BEGIN
   BB_G1.E.Ein := TRUE;
   BB_G1.E.Anst := FALSE;
   BB_G1.E.FU := FALSE;
   BB_G1.E.EA := FALSE;
   BB_G1.E.EZ := FALSE;
   BB_G1.E.MS_St := FALSE;
   BB_G1.E.Th_St := FALSE;
   BB_G1.E.DMA_St := FALSE;
   BB_G1.E.DMZ_St := FALSE;
   BB_G1.E.FU_St := FALSE;
   BB_G1.E.TL_St := FALSE;
   BB_G1.E.UDr_St := FALSE;
   BB_G1.E.UeDr_St := FALSE;
   BB_G1.E.UT_St := FALSE;
   BB_G1.E.Le_St := FALSE;
   BB_G1.E.UeLM_St := FALSE;
   BB_G1.E.UeLE_St := FALSE;
   BB_G1.E.Kom_DP_St := FALSE;
   BB_G1.E.Kom_int_St := FALSE;
   BB_G1.E.int_St := FALSE;
   BB_G1.E.Wart_Wa := FALSE;
   BB_G1.E.Bed_vOrt := FALSE;
   BB_G1.E.Bed_Fern := TRUE;
   BB_G1.E.Bed_UV := FALSE;
   BB_G1.E.Aus := FALSE;
   BB_G1.E.NA := FALSE;
   BB_G1.E.AF_St := FALSE;
   BB_G1.E.Strm := FALSE;
   BB_G1.E.FI_St := FALSE;
   BB_G1.E.SA_St := FALSE;
   BB_G1.E.DD_St := FALSE;
   BB_G1.E.St := FALSE;
   BB_G1.A.Ein := TRUE;
   BB_G1.A.B2 := FALSE;
   BB_G1.A.FU := FALSE;
   BB_G1.A.Req_extern_B1 := TRUE;
   BB_G1.A.Req_extern_B2 := FALSE;
   BB_G1.A.Dir := FALSE;
   BB_G1.A.RST := FALSE;
   BB_G1.A.Auf := FALSE;
   BB_G1.A.Zu := FALSE;
   BB_G1.A.Res9 := FALSE;
   BB_G1.A.Res10 := FALSE;
   BB_G1.A.Res11 := FALSE;
   BB_G1.A.Res12 := FALSE;
   BB_G1.A.Res13 := FALSE;
   BB_G1.A.Res14 := FALSE;
   BB_G1.A.Quit_extern := FALSE;
   BB_G2.E.Ein := TRUE;
   BB_G2.E.Anst := FALSE;
   BB_G2.E.FU := FALSE;
   BB_G2.E.EA := FALSE;
   BB_G2.E.EZ := FALSE;
   BB_G2.E.MS_St := FALSE;
   BB_G2.E.Th_St := FALSE;
   BB_G2.E.DMA_St := FALSE;
   BB_G2.E.DMZ_St := FALSE;
   BB_G2.E.FU_St := FALSE;
   BB_G2.E.TL_St := FALSE;
   BB_G2.E.UDr_St := FALSE;
   BB_G2.E.UeDr_St := FALSE;
   BB_G2.E.UT_St := FALSE;
   BB_G2.E.Le_St := FALSE;
   BB_G2.E.UeLM_St := FALSE;
   BB_G2.E.UeLE_St := FALSE;
   BB_G2.E.Kom_DP_St := FALSE;
   BB_G2.E.Kom_int_St := FALSE;
   BB_G2.E.int_St := FALSE;
   BB_G2.E.Wart_Wa := FALSE;
   BB_G2.E.Bed_vOrt := FALSE;
   BB_G2.E.Bed_Fern := TRUE;
   BB_G2.E.Bed_UV := FALSE;
   BB_G2.E.Aus := FALSE;
   BB_G2.E.NA := FALSE;
   BB_G2.E.AF_St := FALSE;
   BB_G2.E.Strm := FALSE;
   BB_G2.E.FI_St := FALSE;
   BB_G2.E.SA_St := FALSE;
   BB_G2.E.DD_St := FALSE;
   BB_G2.E.St := FALSE;
   BB_G2.A.Ein := TRUE;
   BB_G2.A.B2 := FALSE;
   BB_G2.A.FU := FALSE;
   BB_G2.A.Req_extern_B1 := TRUE;
   BB_G2.A.Req_extern_B2 := FALSE;
   BB_G2.A.Dir := FALSE;
   BB_G2.A.RST := FALSE;
   BB_G2.A.Auf := FALSE;
   BB_G2.A.Zu := FALSE;
   BB_G2.A.Res9 := FALSE;
   BB_G2.A.Res10 := FALSE;
   BB_G2.A.Res11 := FALSE;
   BB_G2.A.Res12 := FALSE;
   BB_G2.A.Res13 := FALSE;
   BB_G2.A.Res14 := FALSE;
   BB_G2.A.Quit_extern := FALSE;
   BB_G3.E.Ein := FALSE;
   BB_G3.E.Anst := FALSE;
   BB_G3.E.FU := FALSE;
   BB_G3.E.EA := FALSE;
   BB_G3.E.EZ := FALSE;
   BB_G3.E.MS_St := FALSE;
   BB_G3.E.Th_St := FALSE;
   BB_G3.E.DMA_St := FALSE;
   BB_G3.E.DMZ_St := FALSE;
   BB_G3.E.FU_St := FALSE;
   BB_G3.E.TL_St := FALSE;
   BB_G3.E.UDr_St := FALSE;
   BB_G3.E.UeDr_St := FALSE;
   BB_G3.E.UT_St := FALSE;
   BB_G3.E.Le_St := FALSE;
   BB_G3.E.UeLM_St := FALSE;
   BB_G3.E.UeLE_St := FALSE;
   BB_G3.E.Kom_DP_St := FALSE;
   BB_G3.E.Kom_int_St := FALSE;
   BB_G3.E.int_St := FALSE;
   BB_G3.E.Wart_Wa := FALSE;
   BB_G3.E.Bed_vOrt := FALSE;
   BB_G3.E.Bed_Fern := TRUE;
   BB_G3.E.Bed_UV := FALSE;
   BB_G3.E.Aus := FALSE;
   BB_G3.E.NA := FALSE;
   BB_G3.E.AF_St := FALSE;
   BB_G3.E.Strm := FALSE;
   BB_G3.E.FI_St := FALSE;
   BB_G3.E.SA_St := FALSE;
   BB_G3.E.DD_St := FALSE;
   BB_G3.E.St := FALSE;
   BB_G3.A.Ein := FALSE;
   BB_G3.A.B2 := FALSE;
   BB_G3.A.FU := FALSE;
   BB_G3.A.Req_extern_B1 := FALSE;
   BB_G3.A.Req_extern_B2 := FALSE;
   BB_G3.A.Dir := FALSE;
   BB_G3.A.RST := FALSE;
   BB_G3.A.Auf := FALSE;
   BB_G3.A.Zu := FALSE;
   BB_G3.A.Res9 := FALSE;
   BB_G3.A.Res10 := FALSE;
   BB_G3.A.Res11 := FALSE;
   BB_G3.A.Res12 := FALSE;
   BB_G3.A.Res13 := FALSE;
   BB_G3.A.Res14 := FALSE;
   BB_G3.A.Quit_extern := FALSE;
   BB_SHL_G1.E.Ein := TRUE;
   BB_SHL_G1.E.Anst := FALSE;
   BB_SHL_G1.E.FU := FALSE;
   BB_SHL_G1.E.EA := FALSE;
   BB_SHL_G1.E.EZ := FALSE;
   BB_SHL_G1.E.MS_St := FALSE;
   BB_SHL_G1.E.Th_St := FALSE;
   BB_SHL_G1.E.DMA_St := FALSE;
   BB_SHL_G1.E.DMZ_St := FALSE;
   BB_SHL_G1.E.FU_St := FALSE;
   BB_SHL_G1.E.TL_St := FALSE;
   BB_SHL_G1.E.UDr_St := FALSE;
   BB_SHL_G1.E.UeDr_St := FALSE;
   BB_SHL_G1.E.UT_St := FALSE;
   BB_SHL_G1.E.Le_St := FALSE;
   BB_SHL_G1.E.UeLM_St := FALSE;
   BB_SHL_G1.E.UeLE_St := FALSE;
   BB_SHL_G1.E.Kom_DP_St := FALSE;
   BB_SHL_G1.E.Kom_int_St := FALSE;
   BB_SHL_G1.E.int_St := FALSE;
   BB_SHL_G1.E.Wart_Wa := FALSE;
   BB_SHL_G1.E.Bed_vOrt := FALSE;
   BB_SHL_G1.E.Bed_Fern := TRUE;
   BB_SHL_G1.E.Bed_UV := FALSE;
   BB_SHL_G1.E.Aus := FALSE;
   BB_SHL_G1.E.NA := FALSE;
   BB_SHL_G1.E.AF_St := FALSE;
   BB_SHL_G1.E.Strm := FALSE;
   BB_SHL_G1.E.FI_St := FALSE;
   BB_SHL_G1.E.SA_St := FALSE;
   BB_SHL_G1.E.DD_St := FALSE;
   BB_SHL_G1.E.St := FALSE;
   BB_SHL_G1.A.Ein := FALSE;
   BB_SHL_G1.A.B2 := FALSE;
   BB_SHL_G1.A.FU := FALSE;
   BB_SHL_G1.A.Req_extern_B1 := FALSE;
   BB_SHL_G1.A.Req_extern_B2 := FALSE;
   BB_SHL_G1.A.Dir := FALSE;
   BB_SHL_G1.A.RST := FALSE;
   BB_SHL_G1.A.Auf := FALSE;
   BB_SHL_G1.A.Zu := FALSE;
   BB_SHL_G1.A.Res9 := FALSE;
   BB_SHL_G1.A.Res10 := FALSE;
   BB_SHL_G1.A.Res11 := FALSE;
   BB_SHL_G1.A.Res12 := FALSE;
   BB_SHL_G1.A.Res13 := FALSE;
   BB_SHL_G1.A.Res14 := FALSE;
   BB_SHL_G1.A.Quit_extern := FALSE;
   BB_SHL_G2.E.Ein := TRUE;
   BB_SHL_G2.E.Anst := FALSE;
   BB_SHL_G2.E.FU := FALSE;
   BB_SHL_G2.E.EA := FALSE;
   BB_SHL_G2.E.EZ := FALSE;
   BB_SHL_G2.E.MS_St := FALSE;
   BB_SHL_G2.E.Th_St := FALSE;
   BB_SHL_G2.E.DMA_St := FALSE;
   BB_SHL_G2.E.DMZ_St := FALSE;
   BB_SHL_G2.E.FU_St := FALSE;
   BB_SHL_G2.E.TL_St := FALSE;
   BB_SHL_G2.E.UDr_St := FALSE;
   BB_SHL_G2.E.UeDr_St := FALSE;
   BB_SHL_G2.E.UT_St := FALSE;
   BB_SHL_G2.E.Le_St := FALSE;
   BB_SHL_G2.E.UeLM_St := FALSE;
   BB_SHL_G2.E.UeLE_St := FALSE;
   BB_SHL_G2.E.Kom_DP_St := FALSE;
   BB_SHL_G2.E.Kom_int_St := FALSE;
   BB_SHL_G2.E.int_St := FALSE;
   BB_SHL_G2.E.Wart_Wa := FALSE;
   BB_SHL_G2.E.Bed_vOrt := FALSE;
   BB_SHL_G2.E.Bed_Fern := TRUE;
   BB_SHL_G2.E.Bed_UV := FALSE;
   BB_SHL_G2.E.Aus := FALSE;
   BB_SHL_G2.E.NA := FALSE;
   BB_SHL_G2.E.AF_St := FALSE;
   BB_SHL_G2.E.Strm := FALSE;
   BB_SHL_G2.E.FI_St := FALSE;
   BB_SHL_G2.E.SA_St := FALSE;
   BB_SHL_G2.E.DD_St := FALSE;
   BB_SHL_G2.E.St := FALSE;
   BB_SHL_G2.A.Ein := FALSE;
   BB_SHL_G2.A.B2 := FALSE;
   BB_SHL_G2.A.FU := FALSE;
   BB_SHL_G2.A.Req_extern_B1 := FALSE;
   BB_SHL_G2.A.Req_extern_B2 := FALSE;
   BB_SHL_G2.A.Dir := FALSE;
   BB_SHL_G2.A.RST := FALSE;
   BB_SHL_G2.A.Auf := FALSE;
   BB_SHL_G2.A.Zu := FALSE;
   BB_SHL_G2.A.Res9 := FALSE;
   BB_SHL_G2.A.Res10 := FALSE;
   BB_SHL_G2.A.Res11 := FALSE;
   BB_SHL_G2.A.Res12 := FALSE;
   BB_SHL_G2.A.Res13 := FALSE;
   BB_SHL_G2.A.Res14 := FALSE;
   BB_SHL_G2.A.Quit_extern := FALSE;
   BB_SHL_G3.E.Ein := FALSE;
   BB_SHL_G3.E.Anst := FALSE;
   BB_SHL_G3.E.FU := FALSE;
   BB_SHL_G3.E.EA := FALSE;
   BB_SHL_G3.E.EZ := FALSE;
   BB_SHL_G3.E.MS_St := FALSE;
   BB_SHL_G3.E.Th_St := FALSE;
   BB_SHL_G3.E.DMA_St := FALSE;
   BB_SHL_G3.E.DMZ_St := FALSE;
   BB_SHL_G3.E.FU_St := FALSE;
   BB_SHL_G3.E.TL_St := FALSE;
   BB_SHL_G3.E.UDr_St := FALSE;
   BB_SHL_G3.E.UeDr_St := FALSE;
   BB_SHL_G3.E.UT_St := FALSE;
   BB_SHL_G3.E.Le_St := FALSE;
   BB_SHL_G3.E.UeLM_St := FALSE;
   BB_SHL_G3.E.UeLE_St := FALSE;
   BB_SHL_G3.E.Kom_DP_St := FALSE;
   BB_SHL_G3.E.Kom_int_St := FALSE;
   BB_SHL_G3.E.int_St := FALSE;
   BB_SHL_G3.E.Wart_Wa := FALSE;
   BB_SHL_G3.E.Bed_vOrt := FALSE;
   BB_SHL_G3.E.Bed_Fern := TRUE;
   BB_SHL_G3.E.Bed_UV := FALSE;
   BB_SHL_G3.E.Aus := FALSE;
   BB_SHL_G3.E.NA := FALSE;
   BB_SHL_G3.E.AF_St := FALSE;
   BB_SHL_G3.E.Strm := FALSE;
   BB_SHL_G3.E.FI_St := FALSE;
   BB_SHL_G3.E.SA_St := FALSE;
   BB_SHL_G3.E.DD_St := FALSE;
   BB_SHL_G3.E.St := FALSE;
   BB_SHL_G3.A.Ein := FALSE;
   BB_SHL_G3.A.B2 := FALSE;
   BB_SHL_G3.A.FU := FALSE;
   BB_SHL_G3.A.Req_extern_B1 := FALSE;
   BB_SHL_G3.A.Req_extern_B2 := FALSE;
   BB_SHL_G3.A.Dir := FALSE;
   BB_SHL_G3.A.RST := FALSE;
   BB_SHL_G3.A.Auf := FALSE;
   BB_SHL_G3.A.Zu := FALSE;
   BB_SHL_G3.A.Res9 := FALSE;
   BB_SHL_G3.A.Res10 := FALSE;
   BB_SHL_G3.A.Res11 := FALSE;
   BB_SHL_G3.A.Res12 := FALSE;
   BB_SHL_G3.A.Res13 := FALSE;
   BB_SHL_G3.A.Res14 := FALSE;
   BB_SHL_G3.A.Quit_extern := FALSE;
   BB_AV.E.Ein := FALSE;
   BB_AV.E.Anst := FALSE;
   BB_AV.E.FU := FALSE;
   BB_AV.E.EA := FALSE;
   BB_AV.E.EZ := FALSE;
   BB_AV.E.MS_St := FALSE;
   BB_AV.E.Th_St := FALSE;
   BB_AV.E.DMA_St := FALSE;
   BB_AV.E.DMZ_St := FALSE;
   BB_AV.E.FU_St := FALSE;
   BB_AV.E.TL_St := FALSE;
   BB_AV.E.UDr_St := FALSE;
   BB_AV.E.UeDr_St := FALSE;
   BB_AV.E.UT_St := FALSE;
   BB_AV.E.Le_St := FALSE;
   BB_AV.E.UeLM_St := FALSE;
   BB_AV.E.UeLE_St := FALSE;
   BB_AV.E.Kom_DP_St := FALSE;
   BB_AV.E.Kom_int_St := FALSE;
   BB_AV.E.int_St := FALSE;
   BB_AV.E.Wart_Wa := FALSE;
   BB_AV.E.Bed_vOrt := FALSE;
   BB_AV.E.Bed_Fern := TRUE;
   BB_AV.E.Bed_UV := FALSE;
   BB_AV.E.Aus := FALSE;
   BB_AV.E.NA := FALSE;
   BB_AV.E.AF_St := FALSE;
   BB_AV.E.Strm := FALSE;
   BB_AV.E.FI_St := FALSE;
   BB_AV.E.SA_St := FALSE;
   BB_AV.E.DD_St := FALSE;
   BB_AV.E.St := FALSE;
   BB_AV.A.Ein := FALSE;
   BB_AV.A.B2 := FALSE;
   BB_AV.A.FU := FALSE;
   BB_AV.A.Req_extern_B1 := FALSE;
   BB_AV.A.Req_extern_B2 := FALSE;
   BB_AV.A.Dir := FALSE;
   BB_AV.A.RST := FALSE;
   BB_AV.A.Auf := FALSE;
   BB_AV.A.Zu := FALSE;
   BB_AV.A.Res9 := FALSE;
   BB_AV.A.Res10 := FALSE;
   BB_AV.A.Res11 := FALSE;
   BB_AV.A.Res12 := FALSE;
   BB_AV.A.Res13 := FALSE;
   BB_AV.A.Res14 := FALSE;
   BB_AV.A.Quit_extern := FALSE;
   BB_LS1.E.Ein := FALSE;
   BB_LS1.E.Anst := FALSE;
   BB_LS1.E.FU := FALSE;
   BB_LS1.E.EA := FALSE;
   BB_LS1.E.EZ := TRUE;
   BB_LS1.E.MS_St := FALSE;
   BB_LS1.E.Th_St := FALSE;
   BB_LS1.E.DMA_St := FALSE;
   BB_LS1.E.DMZ_St := FALSE;
   BB_LS1.E.FU_St := FALSE;
   BB_LS1.E.TL_St := FALSE;
   BB_LS1.E.UDr_St := FALSE;
   BB_LS1.E.UeDr_St := FALSE;
   BB_LS1.E.UT_St := FALSE;
   BB_LS1.E.Le_St := FALSE;
   BB_LS1.E.UeLM_St := FALSE;
   BB_LS1.E.UeLE_St := FALSE;
   BB_LS1.E.Kom_DP_St := FALSE;
   BB_LS1.E.Kom_int_St := FALSE;
   BB_LS1.E.int_St := FALSE;
   BB_LS1.E.Wart_Wa := FALSE;
   BB_LS1.E.Bed_vOrt := FALSE;
   BB_LS1.E.Bed_Fern := TRUE;
   BB_LS1.E.Bed_UV := FALSE;
   BB_LS1.E.Aus := FALSE;
   BB_LS1.E.NA := FALSE;
   BB_LS1.E.AF_St := FALSE;
   BB_LS1.E.Strm := FALSE;
   BB_LS1.E.FI_St := FALSE;
   BB_LS1.E.SA_St := FALSE;
   BB_LS1.E.DD_St := FALSE;
   BB_LS1.E.St := FALSE;
   BB_LS1.A.Ein := FALSE;
   BB_LS1.A.B2 := FALSE;
   BB_LS1.A.FU := FALSE;
   BB_LS1.A.Req_extern_B1 := FALSE;
   BB_LS1.A.Req_extern_B2 := FALSE;
   BB_LS1.A.Dir := FALSE;
   BB_LS1.A.RST := FALSE;
   BB_LS1.A.Auf := FALSE;
   BB_LS1.A.Zu := FALSE;
   BB_LS1.A.Res9 := FALSE;
   BB_LS1.A.Res10 := FALSE;
   BB_LS1.A.Res11 := FALSE;
   BB_LS1.A.Res12 := FALSE;
   BB_LS1.A.Res13 := FALSE;
   BB_LS1.A.Res14 := FALSE;
   BB_LS1.A.Quit_extern := FALSE;
   BB_LS2.E.Ein := FALSE;
   BB_LS2.E.Anst := FALSE;
   BB_LS2.E.FU := FALSE;
   BB_LS2.E.EA := FALSE;
   BB_LS2.E.EZ := TRUE;
   BB_LS2.E.MS_St := FALSE;
   BB_LS2.E.Th_St := FALSE;
   BB_LS2.E.DMA_St := FALSE;
   BB_LS2.E.DMZ_St := FALSE;
   BB_LS2.E.FU_St := FALSE;
   BB_LS2.E.TL_St := FALSE;
   BB_LS2.E.UDr_St := FALSE;
   BB_LS2.E.UeDr_St := FALSE;
   BB_LS2.E.UT_St := FALSE;
   BB_LS2.E.Le_St := FALSE;
   BB_LS2.E.UeLM_St := FALSE;
   BB_LS2.E.UeLE_St := FALSE;
   BB_LS2.E.Kom_DP_St := FALSE;
   BB_LS2.E.Kom_int_St := FALSE;
   BB_LS2.E.int_St := FALSE;
   BB_LS2.E.Wart_Wa := FALSE;
   BB_LS2.E.Bed_vOrt := FALSE;
   BB_LS2.E.Bed_Fern := TRUE;
   BB_LS2.E.Bed_UV := FALSE;
   BB_LS2.E.Aus := FALSE;
   BB_LS2.E.NA := FALSE;
   BB_LS2.E.AF_St := FALSE;
   BB_LS2.E.Strm := FALSE;
   BB_LS2.E.FI_St := FALSE;
   BB_LS2.E.SA_St := FALSE;
   BB_LS2.E.DD_St := FALSE;
   BB_LS2.E.St := FALSE;
   BB_LS2.A.Ein := FALSE;
   BB_LS2.A.B2 := FALSE;
   BB_LS2.A.FU := FALSE;
   BB_LS2.A.Req_extern_B1 := FALSE;
   BB_LS2.A.Req_extern_B2 := FALSE;
   BB_LS2.A.Dir := FALSE;
   BB_LS2.A.RST := FALSE;
   BB_LS2.A.Auf := FALSE;
   BB_LS2.A.Zu := FALSE;
   BB_LS2.A.Res9 := FALSE;
   BB_LS2.A.Res10 := FALSE;
   BB_LS2.A.Res11 := FALSE;
   BB_LS2.A.Res12 := FALSE;
   BB_LS2.A.Res13 := FALSE;
   BB_LS2.A.Res14 := FALSE;
   BB_LS2.A.Quit_extern := FALSE;
   BB1_RZP1.E.Ein := FALSE;
   BB1_RZP1.E.Anst := FALSE;
   BB1_RZP1.E.FU := FALSE;
   BB1_RZP1.E.EA := FALSE;
   BB1_RZP1.E.EZ := FALSE;
   BB1_RZP1.E.MS_St := FALSE;
   BB1_RZP1.E.Th_St := FALSE;
   BB1_RZP1.E.DMA_St := FALSE;
   BB1_RZP1.E.DMZ_St := FALSE;
   BB1_RZP1.E.FU_St := FALSE;
   BB1_RZP1.E.TL_St := FALSE;
   BB1_RZP1.E.UDr_St := FALSE;
   BB1_RZP1.E.UeDr_St := FALSE;
   BB1_RZP1.E.UT_St := FALSE;
   BB1_RZP1.E.Le_St := FALSE;
   BB1_RZP1.E.UeLM_St := FALSE;
   BB1_RZP1.E.UeLE_St := FALSE;
   BB1_RZP1.E.Kom_DP_St := FALSE;
   BB1_RZP1.E.Kom_int_St := FALSE;
   BB1_RZP1.E.int_St := FALSE;
   BB1_RZP1.E.Wart_Wa := FALSE;
   BB1_RZP1.E.Bed_vOrt := FALSE;
   BB1_RZP1.E.Bed_Fern := TRUE;
   BB1_RZP1.E.Bed_UV := FALSE;
   BB1_RZP1.E.Aus := FALSE;
   BB1_RZP1.E.NA := FALSE;
   BB1_RZP1.E.AF_St := FALSE;
   BB1_RZP1.E.Strm := FALSE;
   BB1_RZP1.E.FI_St := FALSE;
   BB1_RZP1.E.SA_St := FALSE;
   BB1_RZP1.E.DD_St := FALSE;
   BB1_RZP1.E.St := FALSE;
   BB1_RZP1.A.Ein := FALSE;
   BB1_RZP1.A.B2 := FALSE;
   BB1_RZP1.A.FU := FALSE;
   BB1_RZP1.A.Req_extern_B1 := FALSE;
   BB1_RZP1.A.Req_extern_B2 := FALSE;
   BB1_RZP1.A.Dir := FALSE;
   BB1_RZP1.A.RST := FALSE;
   BB1_RZP1.A.Auf := FALSE;
   BB1_RZP1.A.Zu := FALSE;
   BB1_RZP1.A.Res9 := FALSE;
   BB1_RZP1.A.Res10 := FALSE;
   BB1_RZP1.A.Res11 := FALSE;
   BB1_RZP1.A.Res12 := FALSE;
   BB1_RZP1.A.Res13 := FALSE;
   BB1_RZP1.A.Res14 := FALSE;
   BB1_RZP1.A.Quit_extern := FALSE;
   BB1_RZP2.E.Ein := FALSE;
   BB1_RZP2.E.Anst := FALSE;
   BB1_RZP2.E.FU := FALSE;
   BB1_RZP2.E.EA := FALSE;
   BB1_RZP2.E.EZ := FALSE;
   BB1_RZP2.E.MS_St := FALSE;
   BB1_RZP2.E.Th_St := FALSE;
   BB1_RZP2.E.DMA_St := FALSE;
   BB1_RZP2.E.DMZ_St := FALSE;
   BB1_RZP2.E.FU_St := FALSE;
   BB1_RZP2.E.TL_St := FALSE;
   BB1_RZP2.E.UDr_St := FALSE;
   BB1_RZP2.E.UeDr_St := FALSE;
   BB1_RZP2.E.UT_St := FALSE;
   BB1_RZP2.E.Le_St := FALSE;
   BB1_RZP2.E.UeLM_St := FALSE;
   BB1_RZP2.E.UeLE_St := FALSE;
   BB1_RZP2.E.Kom_DP_St := FALSE;
   BB1_RZP2.E.Kom_int_St := FALSE;
   BB1_RZP2.E.int_St := FALSE;
   BB1_RZP2.E.Wart_Wa := FALSE;
   BB1_RZP2.E.Bed_vOrt := FALSE;
   BB1_RZP2.E.Bed_Fern := TRUE;
   BB1_RZP2.E.Bed_UV := FALSE;
   BB1_RZP2.E.Aus := FALSE;
   BB1_RZP2.E.NA := FALSE;
   BB1_RZP2.E.AF_St := FALSE;
   BB1_RZP2.E.Strm := FALSE;
   BB1_RZP2.E.FI_St := FALSE;
   BB1_RZP2.E.SA_St := FALSE;
   BB1_RZP2.E.DD_St := FALSE;
   BB1_RZP2.E.St := FALSE;
   BB1_RZP2.A.Ein := FALSE;
   BB1_RZP2.A.B2 := FALSE;
   BB1_RZP2.A.FU := FALSE;
   BB1_RZP2.A.Req_extern_B1 := FALSE;
   BB1_RZP2.A.Req_extern_B2 := FALSE;
   BB1_RZP2.A.Dir := FALSE;
   BB1_RZP2.A.RST := FALSE;
   BB1_RZP2.A.Auf := FALSE;
   BB1_RZP2.A.Zu := FALSE;
   BB1_RZP2.A.Res9 := FALSE;
   BB1_RZP2.A.Res10 := FALSE;
   BB1_RZP2.A.Res11 := FALSE;
   BB1_RZP2.A.Res12 := FALSE;
   BB1_RZP2.A.Res13 := FALSE;
   BB1_RZP2.A.Res14 := FALSE;
   BB1_RZP2.A.Quit_extern := FALSE;
   BB1_UeSP.E.Ein := FALSE;
   BB1_UeSP.E.Anst := FALSE;
   BB1_UeSP.E.FU := FALSE;
   BB1_UeSP.E.EA := FALSE;
   BB1_UeSP.E.EZ := FALSE;
   BB1_UeSP.E.MS_St := FALSE;
   BB1_UeSP.E.Th_St := FALSE;
   BB1_UeSP.E.DMA_St := FALSE;
   BB1_UeSP.E.DMZ_St := FALSE;
   BB1_UeSP.E.FU_St := FALSE;
   BB1_UeSP.E.TL_St := FALSE;
   BB1_UeSP.E.UDr_St := FALSE;
   BB1_UeSP.E.UeDr_St := FALSE;
   BB1_UeSP.E.UT_St := FALSE;
   BB1_UeSP.E.Le_St := FALSE;
   BB1_UeSP.E.UeLM_St := FALSE;
   BB1_UeSP.E.UeLE_St := FALSE;
   BB1_UeSP.E.Kom_DP_St := FALSE;
   BB1_UeSP.E.Kom_int_St := FALSE;
   BB1_UeSP.E.int_St := FALSE;
   BB1_UeSP.E.Wart_Wa := FALSE;
   BB1_UeSP.E.Bed_vOrt := FALSE;
   BB1_UeSP.E.Bed_Fern := TRUE;
   BB1_UeSP.E.Bed_UV := FALSE;
   BB1_UeSP.E.Aus := FALSE;
   BB1_UeSP.E.NA := FALSE;
   BB1_UeSP.E.AF_St := FALSE;
   BB1_UeSP.E.Strm := FALSE;
   BB1_UeSP.E.FI_St := FALSE;
   BB1_UeSP.E.SA_St := FALSE;
   BB1_UeSP.E.DD_St := FALSE;
   BB1_UeSP.E.St := FALSE;
   BB1_UeSP.A.Ein := FALSE;
   BB1_UeSP.A.B2 := FALSE;
   BB1_UeSP.A.FU := FALSE;
   BB1_UeSP.A.Req_extern_B1 := FALSE;
   BB1_UeSP.A.Req_extern_B2 := FALSE;
   BB1_UeSP.A.Dir := FALSE;
   BB1_UeSP.A.RST := FALSE;
   BB1_UeSP.A.Auf := FALSE;
   BB1_UeSP.A.Zu := FALSE;
   BB1_UeSP.A.Res9 := FALSE;
   BB1_UeSP.A.Res10 := FALSE;
   BB1_UeSP.A.Res11 := FALSE;
   BB1_UeSP.A.Res12 := FALSE;
   BB1_UeSP.A.Res13 := FALSE;
   BB1_UeSP.A.Res14 := FALSE;
   BB1_UeSP.A.Quit_extern := FALSE;
   BB1_AS1.E.Ein := FALSE;
   BB1_AS1.E.Anst := FALSE;
   BB1_AS1.E.FU := FALSE;
   BB1_AS1.E.EA := TRUE;
   BB1_AS1.E.EZ := FALSE;
   BB1_AS1.E.MS_St := FALSE;
   BB1_AS1.E.Th_St := FALSE;
   BB1_AS1.E.DMA_St := FALSE;
   BB1_AS1.E.DMZ_St := FALSE;
   BB1_AS1.E.FU_St := FALSE;
   BB1_AS1.E.TL_St := FALSE;
   BB1_AS1.E.UDr_St := FALSE;
   BB1_AS1.E.UeDr_St := FALSE;
   BB1_AS1.E.UT_St := FALSE;
   BB1_AS1.E.Le_St := FALSE;
   BB1_AS1.E.UeLM_St := FALSE;
   BB1_AS1.E.UeLE_St := FALSE;
   BB1_AS1.E.Kom_DP_St := FALSE;
   BB1_AS1.E.Kom_int_St := FALSE;
   BB1_AS1.E.int_St := FALSE;
   BB1_AS1.E.Wart_Wa := FALSE;
   BB1_AS1.E.Bed_vOrt := FALSE;
   BB1_AS1.E.Bed_Fern := TRUE;
   BB1_AS1.E.Bed_UV := FALSE;
   BB1_AS1.E.Aus := FALSE;
   BB1_AS1.E.NA := FALSE;
   BB1_AS1.E.AF_St := FALSE;
   BB1_AS1.E.Strm := FALSE;
   BB1_AS1.E.FI_St := FALSE;
   BB1_AS1.E.SA_St := FALSE;
   BB1_AS1.E.DD_St := FALSE;
   BB1_AS1.E.St := FALSE;
   BB1_AS1.A.Ein := FALSE;
   BB1_AS1.A.B2 := FALSE;
   BB1_AS1.A.FU := FALSE;
   BB1_AS1.A.Req_extern_B1 := FALSE;
   BB1_AS1.A.Req_extern_B2 := FALSE;
   BB1_AS1.A.Dir := FALSE;
   BB1_AS1.A.RST := FALSE;
   BB1_AS1.A.Auf := FALSE;
   BB1_AS1.A.Zu := FALSE;
   BB1_AS1.A.Res9 := FALSE;
   BB1_AS1.A.Res10 := FALSE;
   BB1_AS1.A.Res11 := FALSE;
   BB1_AS1.A.Res12 := FALSE;
   BB1_AS1.A.Res13 := FALSE;
   BB1_AS1.A.Res14 := FALSE;
   BB1_AS1.A.Quit_extern := FALSE;
   BB1_AS2.E.Ein := FALSE;
   BB1_AS2.E.Anst := FALSE;
   BB1_AS2.E.FU := FALSE;
   BB1_AS2.E.EA := FALSE;
   BB1_AS2.E.EZ := TRUE;
   BB1_AS2.E.MS_St := FALSE;
   BB1_AS2.E.Th_St := FALSE;
   BB1_AS2.E.DMA_St := FALSE;
   BB1_AS2.E.DMZ_St := FALSE;
   BB1_AS2.E.FU_St := FALSE;
   BB1_AS2.E.TL_St := FALSE;
   BB1_AS2.E.UDr_St := FALSE;
   BB1_AS2.E.UeDr_St := FALSE;
   BB1_AS2.E.UT_St := FALSE;
   BB1_AS2.E.Le_St := FALSE;
   BB1_AS2.E.UeLM_St := FALSE;
   BB1_AS2.E.UeLE_St := FALSE;
   BB1_AS2.E.Kom_DP_St := FALSE;
   BB1_AS2.E.Kom_int_St := FALSE;
   BB1_AS2.E.int_St := FALSE;
   BB1_AS2.E.Wart_Wa := FALSE;
   BB1_AS2.E.Bed_vOrt := FALSE;
   BB1_AS2.E.Bed_Fern := TRUE;
   BB1_AS2.E.Bed_UV := FALSE;
   BB1_AS2.E.Aus := FALSE;
   BB1_AS2.E.NA := FALSE;
   BB1_AS2.E.AF_St := FALSE;
   BB1_AS2.E.Strm := FALSE;
   BB1_AS2.E.FI_St := FALSE;
   BB1_AS2.E.SA_St := FALSE;
   BB1_AS2.E.DD_St := FALSE;
   BB1_AS2.E.St := FALSE;
   BB1_AS2.A.Ein := FALSE;
   BB1_AS2.A.B2 := FALSE;
   BB1_AS2.A.FU := FALSE;
   BB1_AS2.A.Req_extern_B1 := FALSE;
   BB1_AS2.A.Req_extern_B2 := FALSE;
   BB1_AS2.A.Dir := FALSE;
   BB1_AS2.A.RST := FALSE;
   BB1_AS2.A.Auf := FALSE;
   BB1_AS2.A.Zu := FALSE;
   BB1_AS2.A.Res9 := FALSE;
   BB1_AS2.A.Res10 := FALSE;
   BB1_AS2.A.Res11 := FALSE;
   BB1_AS2.A.Res12 := FALSE;
   BB1_AS2.A.Res13 := FALSE;
   BB1_AS2.A.Res14 := FALSE;
   BB1_AS2.A.Quit_extern := FALSE;
   BB1_SR1.E.Ein := FALSE;
   BB1_SR1.E.Anst := FALSE;
   BB1_SR1.E.FU := FALSE;
   BB1_SR1.E.EA := FALSE;
   BB1_SR1.E.EZ := FALSE;
   BB1_SR1.E.MS_St := FALSE;
   BB1_SR1.E.Th_St := FALSE;
   BB1_SR1.E.DMA_St := FALSE;
   BB1_SR1.E.DMZ_St := FALSE;
   BB1_SR1.E.FU_St := FALSE;
   BB1_SR1.E.TL_St := FALSE;
   BB1_SR1.E.UDr_St := FALSE;
   BB1_SR1.E.UeDr_St := FALSE;
   BB1_SR1.E.UT_St := FALSE;
   BB1_SR1.E.Le_St := FALSE;
   BB1_SR1.E.UeLM_St := FALSE;
   BB1_SR1.E.UeLE_St := FALSE;
   BB1_SR1.E.Kom_DP_St := FALSE;
   BB1_SR1.E.Kom_int_St := FALSE;
   BB1_SR1.E.int_St := FALSE;
   BB1_SR1.E.Wart_Wa := FALSE;
   BB1_SR1.E.Bed_vOrt := FALSE;
   BB1_SR1.E.Bed_Fern := TRUE;
   BB1_SR1.E.Bed_UV := FALSE;
   BB1_SR1.E.Aus := FALSE;
   BB1_SR1.E.NA := FALSE;
   BB1_SR1.E.AF_St := FALSE;
   BB1_SR1.E.Strm := FALSE;
   BB1_SR1.E.FI_St := FALSE;
   BB1_SR1.E.SA_St := FALSE;
   BB1_SR1.E.DD_St := FALSE;
   BB1_SR1.E.St := FALSE;
   BB1_SR1.A.Ein := FALSE;
   BB1_SR1.A.B2 := FALSE;
   BB1_SR1.A.FU := FALSE;
   BB1_SR1.A.Req_extern_B1 := FALSE;
   BB1_SR1.A.Req_extern_B2 := FALSE;
   BB1_SR1.A.Dir := FALSE;
   BB1_SR1.A.RST := FALSE;
   BB1_SR1.A.Auf := FALSE;
   BB1_SR1.A.Zu := FALSE;
   BB1_SR1.A.Res9 := FALSE;
   BB1_SR1.A.Res10 := FALSE;
   BB1_SR1.A.Res11 := FALSE;
   BB1_SR1.A.Res12 := FALSE;
   BB1_SR1.A.Res13 := FALSE;
   BB1_SR1.A.Res14 := FALSE;
   BB1_SR1.A.Quit_extern := FALSE;
   BB1_SR2.E.Ein := FALSE;
   BB1_SR2.E.Anst := FALSE;
   BB1_SR2.E.FU := FALSE;
   BB1_SR2.E.EA := FALSE;
   BB1_SR2.E.EZ := FALSE;
   BB1_SR2.E.MS_St := FALSE;
   BB1_SR2.E.Th_St := FALSE;
   BB1_SR2.E.DMA_St := FALSE;
   BB1_SR2.E.DMZ_St := FALSE;
   BB1_SR2.E.FU_St := FALSE;
   BB1_SR2.E.TL_St := FALSE;
   BB1_SR2.E.UDr_St := FALSE;
   BB1_SR2.E.UeDr_St := FALSE;
   BB1_SR2.E.UT_St := FALSE;
   BB1_SR2.E.Le_St := FALSE;
   BB1_SR2.E.UeLM_St := FALSE;
   BB1_SR2.E.UeLE_St := FALSE;
   BB1_SR2.E.Kom_DP_St := FALSE;
   BB1_SR2.E.Kom_int_St := FALSE;
   BB1_SR2.E.int_St := FALSE;
   BB1_SR2.E.Wart_Wa := FALSE;
   BB1_SR2.E.Bed_vOrt := FALSE;
   BB1_SR2.E.Bed_Fern := TRUE;
   BB1_SR2.E.Bed_UV := FALSE;
   BB1_SR2.E.Aus := FALSE;
   BB1_SR2.E.NA := FALSE;
   BB1_SR2.E.AF_St := FALSE;
   BB1_SR2.E.Strm := FALSE;
   BB1_SR2.E.FI_St := FALSE;
   BB1_SR2.E.SA_St := FALSE;
   BB1_SR2.E.DD_St := FALSE;
   BB1_SR2.E.St := FALSE;
   BB1_SR2.A.Ein := FALSE;
   BB1_SR2.A.B2 := FALSE;
   BB1_SR2.A.FU := FALSE;
   BB1_SR2.A.Req_extern_B1 := FALSE;
   BB1_SR2.A.Req_extern_B2 := FALSE;
   BB1_SR2.A.Dir := FALSE;
   BB1_SR2.A.RST := FALSE;
   BB1_SR2.A.Auf := FALSE;
   BB1_SR2.A.Zu := FALSE;
   BB1_SR2.A.Res9 := FALSE;
   BB1_SR2.A.Res10 := FALSE;
   BB1_SR2.A.Res11 := FALSE;
   BB1_SR2.A.Res12 := FALSE;
   BB1_SR2.A.Res13 := FALSE;
   BB1_SR2.A.Res14 := FALSE;
   BB1_SR2.A.Quit_extern := FALSE;
   BB2_RZP1.E.Ein := FALSE;
   BB2_RZP1.E.Anst := FALSE;
   BB2_RZP1.E.FU := FALSE;
   BB2_RZP1.E.EA := FALSE;
   BB2_RZP1.E.EZ := FALSE;
   BB2_RZP1.E.MS_St := FALSE;
   BB2_RZP1.E.Th_St := FALSE;
   BB2_RZP1.E.DMA_St := FALSE;
   BB2_RZP1.E.DMZ_St := FALSE;
   BB2_RZP1.E.FU_St := FALSE;
   BB2_RZP1.E.TL_St := FALSE;
   BB2_RZP1.E.UDr_St := FALSE;
   BB2_RZP1.E.UeDr_St := FALSE;
   BB2_RZP1.E.UT_St := FALSE;
   BB2_RZP1.E.Le_St := FALSE;
   BB2_RZP1.E.UeLM_St := FALSE;
   BB2_RZP1.E.UeLE_St := FALSE;
   BB2_RZP1.E.Kom_DP_St := FALSE;
   BB2_RZP1.E.Kom_int_St := FALSE;
   BB2_RZP1.E.int_St := FALSE;
   BB2_RZP1.E.Wart_Wa := FALSE;
   BB2_RZP1.E.Bed_vOrt := FALSE;
   BB2_RZP1.E.Bed_Fern := TRUE;
   BB2_RZP1.E.Bed_UV := FALSE;
   BB2_RZP1.E.Aus := FALSE;
   BB2_RZP1.E.NA := FALSE;
   BB2_RZP1.E.AF_St := FALSE;
   BB2_RZP1.E.Strm := FALSE;
   BB2_RZP1.E.FI_St := FALSE;
   BB2_RZP1.E.SA_St := FALSE;
   BB2_RZP1.E.DD_St := FALSE;
   BB2_RZP1.E.St := FALSE;
   BB2_RZP1.A.Ein := FALSE;
   BB2_RZP1.A.B2 := FALSE;
   BB2_RZP1.A.FU := FALSE;
   BB2_RZP1.A.Req_extern_B1 := FALSE;
   BB2_RZP1.A.Req_extern_B2 := FALSE;
   BB2_RZP1.A.Dir := FALSE;
   BB2_RZP1.A.RST := FALSE;
   BB2_RZP1.A.Auf := FALSE;
   BB2_RZP1.A.Zu := FALSE;
   BB2_RZP1.A.Res9 := FALSE;
   BB2_RZP1.A.Res10 := FALSE;
   BB2_RZP1.A.Res11 := FALSE;
   BB2_RZP1.A.Res12 := FALSE;
   BB2_RZP1.A.Res13 := FALSE;
   BB2_RZP1.A.Res14 := FALSE;
   BB2_RZP1.A.Quit_extern := FALSE;
   BB2_RZP2.E.Ein := FALSE;
   BB2_RZP2.E.Anst := FALSE;
   BB2_RZP2.E.FU := FALSE;
   BB2_RZP2.E.EA := FALSE;
   BB2_RZP2.E.EZ := FALSE;
   BB2_RZP2.E.MS_St := FALSE;
   BB2_RZP2.E.Th_St := FALSE;
   BB2_RZP2.E.DMA_St := FALSE;
   BB2_RZP2.E.DMZ_St := FALSE;
   BB2_RZP2.E.FU_St := FALSE;
   BB2_RZP2.E.TL_St := FALSE;
   BB2_RZP2.E.UDr_St := FALSE;
   BB2_RZP2.E.UeDr_St := FALSE;
   BB2_RZP2.E.UT_St := FALSE;
   BB2_RZP2.E.Le_St := FALSE;
   BB2_RZP2.E.UeLM_St := FALSE;
   BB2_RZP2.E.UeLE_St := FALSE;
   BB2_RZP2.E.Kom_DP_St := FALSE;
   BB2_RZP2.E.Kom_int_St := FALSE;
   BB2_RZP2.E.int_St := FALSE;
   BB2_RZP2.E.Wart_Wa := FALSE;
   BB2_RZP2.E.Bed_vOrt := FALSE;
   BB2_RZP2.E.Bed_Fern := TRUE;
   BB2_RZP2.E.Bed_UV := FALSE;
   BB2_RZP2.E.Aus := FALSE;
   BB2_RZP2.E.NA := FALSE;
   BB2_RZP2.E.AF_St := FALSE;
   BB2_RZP2.E.Strm := FALSE;
   BB2_RZP2.E.FI_St := FALSE;
   BB2_RZP2.E.SA_St := FALSE;
   BB2_RZP2.E.DD_St := FALSE;
   BB2_RZP2.E.St := FALSE;
   BB2_RZP2.A.Ein := FALSE;
   BB2_RZP2.A.B2 := FALSE;
   BB2_RZP2.A.FU := FALSE;
   BB2_RZP2.A.Req_extern_B1 := FALSE;
   BB2_RZP2.A.Req_extern_B2 := FALSE;
   BB2_RZP2.A.Dir := FALSE;
   BB2_RZP2.A.RST := FALSE;
   BB2_RZP2.A.Auf := FALSE;
   BB2_RZP2.A.Zu := FALSE;
   BB2_RZP2.A.Res9 := FALSE;
   BB2_RZP2.A.Res10 := FALSE;
   BB2_RZP2.A.Res11 := FALSE;
   BB2_RZP2.A.Res12 := FALSE;
   BB2_RZP2.A.Res13 := FALSE;
   BB2_RZP2.A.Res14 := FALSE;
   BB2_RZP2.A.Quit_extern := FALSE;
   BB2_UeSP.E.Ein := FALSE;
   BB2_UeSP.E.Anst := FALSE;
   BB2_UeSP.E.FU := FALSE;
   BB2_UeSP.E.EA := FALSE;
   BB2_UeSP.E.EZ := FALSE;
   BB2_UeSP.E.MS_St := FALSE;
   BB2_UeSP.E.Th_St := FALSE;
   BB2_UeSP.E.DMA_St := FALSE;
   BB2_UeSP.E.DMZ_St := FALSE;
   BB2_UeSP.E.FU_St := FALSE;
   BB2_UeSP.E.TL_St := FALSE;
   BB2_UeSP.E.UDr_St := FALSE;
   BB2_UeSP.E.UeDr_St := FALSE;
   BB2_UeSP.E.UT_St := FALSE;
   BB2_UeSP.E.Le_St := FALSE;
   BB2_UeSP.E.UeLM_St := FALSE;
   BB2_UeSP.E.UeLE_St := FALSE;
   BB2_UeSP.E.Kom_DP_St := FALSE;
   BB2_UeSP.E.Kom_int_St := FALSE;
   BB2_UeSP.E.int_St := FALSE;
   BB2_UeSP.E.Wart_Wa := FALSE;
   BB2_UeSP.E.Bed_vOrt := FALSE;
   BB2_UeSP.E.Bed_Fern := TRUE;
   BB2_UeSP.E.Bed_UV := FALSE;
   BB2_UeSP.E.Aus := FALSE;
   BB2_UeSP.E.NA := FALSE;
   BB2_UeSP.E.AF_St := FALSE;
   BB2_UeSP.E.Strm := FALSE;
   BB2_UeSP.E.FI_St := FALSE;
   BB2_UeSP.E.SA_St := FALSE;
   BB2_UeSP.E.DD_St := FALSE;
   BB2_UeSP.E.St := FALSE;
   BB2_UeSP.A.Ein := FALSE;
   BB2_UeSP.A.B2 := FALSE;
   BB2_UeSP.A.FU := FALSE;
   BB2_UeSP.A.Req_extern_B1 := FALSE;
   BB2_UeSP.A.Req_extern_B2 := FALSE;
   BB2_UeSP.A.Dir := FALSE;
   BB2_UeSP.A.RST := FALSE;
   BB2_UeSP.A.Auf := FALSE;
   BB2_UeSP.A.Zu := FALSE;
   BB2_UeSP.A.Res9 := FALSE;
   BB2_UeSP.A.Res10 := FALSE;
   BB2_UeSP.A.Res11 := FALSE;
   BB2_UeSP.A.Res12 := FALSE;
   BB2_UeSP.A.Res13 := FALSE;
   BB2_UeSP.A.Res14 := FALSE;
   BB2_UeSP.A.Quit_extern := FALSE;
   BB2_AS1.E.Ein := FALSE;
   BB2_AS1.E.Anst := FALSE;
   BB2_AS1.E.FU := FALSE;
   BB2_AS1.E.EA := FALSE;
   BB2_AS1.E.EZ := TRUE;
   BB2_AS1.E.MS_St := FALSE;
   BB2_AS1.E.Th_St := FALSE;
   BB2_AS1.E.DMA_St := FALSE;
   BB2_AS1.E.DMZ_St := FALSE;
   BB2_AS1.E.FU_St := FALSE;
   BB2_AS1.E.TL_St := FALSE;
   BB2_AS1.E.UDr_St := FALSE;
   BB2_AS1.E.UeDr_St := FALSE;
   BB2_AS1.E.UT_St := FALSE;
   BB2_AS1.E.Le_St := FALSE;
   BB2_AS1.E.UeLM_St := FALSE;
   BB2_AS1.E.UeLE_St := FALSE;
   BB2_AS1.E.Kom_DP_St := FALSE;
   BB2_AS1.E.Kom_int_St := FALSE;
   BB2_AS1.E.int_St := FALSE;
   BB2_AS1.E.Wart_Wa := FALSE;
   BB2_AS1.E.Bed_vOrt := FALSE;
   BB2_AS1.E.Bed_Fern := TRUE;
   BB2_AS1.E.Bed_UV := FALSE;
   BB2_AS1.E.Aus := FALSE;
   BB2_AS1.E.NA := FALSE;
   BB2_AS1.E.AF_St := FALSE;
   BB2_AS1.E.Strm := FALSE;
   BB2_AS1.E.FI_St := FALSE;
   BB2_AS1.E.SA_St := FALSE;
   BB2_AS1.E.DD_St := FALSE;
   BB2_AS1.E.St := FALSE;
   BB2_AS1.A.Ein := FALSE;
   BB2_AS1.A.B2 := FALSE;
   BB2_AS1.A.FU := FALSE;
   BB2_AS1.A.Req_extern_B1 := FALSE;
   BB2_AS1.A.Req_extern_B2 := FALSE;
   BB2_AS1.A.Dir := FALSE;
   BB2_AS1.A.RST := FALSE;
   BB2_AS1.A.Auf := FALSE;
   BB2_AS1.A.Zu := FALSE;
   BB2_AS1.A.Res9 := FALSE;
   BB2_AS1.A.Res10 := FALSE;
   BB2_AS1.A.Res11 := FALSE;
   BB2_AS1.A.Res12 := FALSE;
   BB2_AS1.A.Res13 := FALSE;
   BB2_AS1.A.Res14 := FALSE;
   BB2_AS1.A.Quit_extern := FALSE;
   BB2_AS2.E.Ein := FALSE;
   BB2_AS2.E.Anst := FALSE;
   BB2_AS2.E.FU := FALSE;
   BB2_AS2.E.EA := TRUE;
   BB2_AS2.E.EZ := FALSE;
   BB2_AS2.E.MS_St := FALSE;
   BB2_AS2.E.Th_St := FALSE;
   BB2_AS2.E.DMA_St := FALSE;
   BB2_AS2.E.DMZ_St := FALSE;
   BB2_AS2.E.FU_St := FALSE;
   BB2_AS2.E.TL_St := FALSE;
   BB2_AS2.E.UDr_St := FALSE;
   BB2_AS2.E.UeDr_St := FALSE;
   BB2_AS2.E.UT_St := FALSE;
   BB2_AS2.E.Le_St := FALSE;
   BB2_AS2.E.UeLM_St := FALSE;
   BB2_AS2.E.UeLE_St := FALSE;
   BB2_AS2.E.Kom_DP_St := FALSE;
   BB2_AS2.E.Kom_int_St := FALSE;
   BB2_AS2.E.int_St := FALSE;
   BB2_AS2.E.Wart_Wa := FALSE;
   BB2_AS2.E.Bed_vOrt := FALSE;
   BB2_AS2.E.Bed_Fern := TRUE;
   BB2_AS2.E.Bed_UV := FALSE;
   BB2_AS2.E.Aus := FALSE;
   BB2_AS2.E.NA := FALSE;
   BB2_AS2.E.AF_St := FALSE;
   BB2_AS2.E.Strm := FALSE;
   BB2_AS2.E.FI_St := FALSE;
   BB2_AS2.E.SA_St := FALSE;
   BB2_AS2.E.DD_St := FALSE;
   BB2_AS2.E.St := FALSE;
   BB2_AS2.A.Ein := FALSE;
   BB2_AS2.A.B2 := FALSE;
   BB2_AS2.A.FU := FALSE;
   BB2_AS2.A.Req_extern_B1 := FALSE;
   BB2_AS2.A.Req_extern_B2 := FALSE;
   BB2_AS2.A.Dir := FALSE;
   BB2_AS2.A.RST := FALSE;
   BB2_AS2.A.Auf := FALSE;
   BB2_AS2.A.Zu := FALSE;
   BB2_AS2.A.Res9 := FALSE;
   BB2_AS2.A.Res10 := FALSE;
   BB2_AS2.A.Res11 := FALSE;
   BB2_AS2.A.Res12 := FALSE;
   BB2_AS2.A.Res13 := FALSE;
   BB2_AS2.A.Res14 := FALSE;
   BB2_AS2.A.Quit_extern := FALSE;
   BB2_SR1.E.Ein := FALSE;
   BB2_SR1.E.Anst := FALSE;
   BB2_SR1.E.FU := FALSE;
   BB2_SR1.E.EA := FALSE;
   BB2_SR1.E.EZ := FALSE;
   BB2_SR1.E.MS_St := FALSE;
   BB2_SR1.E.Th_St := FALSE;
   BB2_SR1.E.DMA_St := FALSE;
   BB2_SR1.E.DMZ_St := FALSE;
   BB2_SR1.E.FU_St := FALSE;
   BB2_SR1.E.TL_St := FALSE;
   BB2_SR1.E.UDr_St := FALSE;
   BB2_SR1.E.UeDr_St := FALSE;
   BB2_SR1.E.UT_St := FALSE;
   BB2_SR1.E.Le_St := FALSE;
   BB2_SR1.E.UeLM_St := FALSE;
   BB2_SR1.E.UeLE_St := FALSE;
   BB2_SR1.E.Kom_DP_St := FALSE;
   BB2_SR1.E.Kom_int_St := FALSE;
   BB2_SR1.E.int_St := FALSE;
   BB2_SR1.E.Wart_Wa := FALSE;
   BB2_SR1.E.Bed_vOrt := FALSE;
   BB2_SR1.E.Bed_Fern := TRUE;
   BB2_SR1.E.Bed_UV := FALSE;
   BB2_SR1.E.Aus := FALSE;
   BB2_SR1.E.NA := FALSE;
   BB2_SR1.E.AF_St := FALSE;
   BB2_SR1.E.Strm := FALSE;
   BB2_SR1.E.FI_St := FALSE;
   BB2_SR1.E.SA_St := FALSE;
   BB2_SR1.E.DD_St := FALSE;
   BB2_SR1.E.St := FALSE;
   BB2_SR1.A.Ein := FALSE;
   BB2_SR1.A.B2 := FALSE;
   BB2_SR1.A.FU := FALSE;
   BB2_SR1.A.Req_extern_B1 := FALSE;
   BB2_SR1.A.Req_extern_B2 := FALSE;
   BB2_SR1.A.Dir := FALSE;
   BB2_SR1.A.RST := FALSE;
   BB2_SR1.A.Auf := FALSE;
   BB2_SR1.A.Zu := FALSE;
   BB2_SR1.A.Res9 := FALSE;
   BB2_SR1.A.Res10 := FALSE;
   BB2_SR1.A.Res11 := FALSE;
   BB2_SR1.A.Res12 := FALSE;
   BB2_SR1.A.Res13 := FALSE;
   BB2_SR1.A.Res14 := FALSE;
   BB2_SR1.A.Quit_extern := FALSE;
   BB2_SR2.E.Ein := FALSE;
   BB2_SR2.E.Anst := FALSE;
   BB2_SR2.E.FU := FALSE;
   BB2_SR2.E.EA := FALSE;
   BB2_SR2.E.EZ := FALSE;
   BB2_SR2.E.MS_St := FALSE;
   BB2_SR2.E.Th_St := FALSE;
   BB2_SR2.E.DMA_St := FALSE;
   BB2_SR2.E.DMZ_St := FALSE;
   BB2_SR2.E.FU_St := FALSE;
   BB2_SR2.E.TL_St := FALSE;
   BB2_SR2.E.UDr_St := FALSE;
   BB2_SR2.E.UeDr_St := FALSE;
   BB2_SR2.E.UT_St := FALSE;
   BB2_SR2.E.Le_St := FALSE;
   BB2_SR2.E.UeLM_St := FALSE;
   BB2_SR2.E.UeLE_St := FALSE;
   BB2_SR2.E.Kom_DP_St := FALSE;
   BB2_SR2.E.Kom_int_St := FALSE;
   BB2_SR2.E.int_St := FALSE;
   BB2_SR2.E.Wart_Wa := FALSE;
   BB2_SR2.E.Bed_vOrt := FALSE;
   BB2_SR2.E.Bed_Fern := TRUE;
   BB2_SR2.E.Bed_UV := FALSE;
   BB2_SR2.E.Aus := FALSE;
   BB2_SR2.E.NA := FALSE;
   BB2_SR2.E.AF_St := FALSE;
   BB2_SR2.E.Strm := FALSE;
   BB2_SR2.E.FI_St := FALSE;
   BB2_SR2.E.SA_St := FALSE;
   BB2_SR2.E.DD_St := FALSE;
   BB2_SR2.E.St := FALSE;
   BB2_SR2.A.Ein := FALSE;
   BB2_SR2.A.B2 := FALSE;
   BB2_SR2.A.FU := FALSE;
   BB2_SR2.A.Req_extern_B1 := FALSE;
   BB2_SR2.A.Req_extern_B2 := FALSE;
   BB2_SR2.A.Dir := FALSE;
   BB2_SR2.A.RST := FALSE;
   BB2_SR2.A.Auf := FALSE;
   BB2_SR2.A.Zu := FALSE;
   BB2_SR2.A.Res9 := FALSE;
   BB2_SR2.A.Res10 := FALSE;
   BB2_SR2.A.Res11 := FALSE;
   BB2_SR2.A.Res12 := FALSE;
   BB2_SR2.A.Res13 := FALSE;
   BB2_SR2.A.Res14 := FALSE;
   BB2_SR2.A.Quit_extern := FALSE;
   BB1_SR_K.E.Ein := FALSE;
   BB1_SR_K.E.Anst := FALSE;
   BB1_SR_K.E.FU := FALSE;
   BB1_SR_K.E.EA := FALSE;
   BB1_SR_K.E.EZ := FALSE;
   BB1_SR_K.E.MS_St := FALSE;
   BB1_SR_K.E.Th_St := FALSE;
   BB1_SR_K.E.DMA_St := FALSE;
   BB1_SR_K.E.DMZ_St := FALSE;
   BB1_SR_K.E.FU_St := FALSE;
   BB1_SR_K.E.TL_St := FALSE;
   BB1_SR_K.E.UDr_St := FALSE;
   BB1_SR_K.E.UeDr_St := FALSE;
   BB1_SR_K.E.UT_St := FALSE;
   BB1_SR_K.E.Le_St := FALSE;
   BB1_SR_K.E.UeLM_St := FALSE;
   BB1_SR_K.E.UeLE_St := FALSE;
   BB1_SR_K.E.Kom_DP_St := FALSE;
   BB1_SR_K.E.Kom_int_St := FALSE;
   BB1_SR_K.E.int_St := FALSE;
   BB1_SR_K.E.Wart_Wa := FALSE;
   BB1_SR_K.E.Bed_vOrt := FALSE;
   BB1_SR_K.E.Bed_Fern := TRUE;
   BB1_SR_K.E.Bed_UV := FALSE;
   BB1_SR_K.E.Aus := FALSE;
   BB1_SR_K.E.NA := FALSE;
   BB1_SR_K.E.AF_St := FALSE;
   BB1_SR_K.E.Strm := FALSE;
   BB1_SR_K.E.FI_St := FALSE;
   BB1_SR_K.E.SA_St := FALSE;
   BB1_SR_K.E.DD_St := FALSE;
   BB1_SR_K.E.St := FALSE;
   BB1_SR_K.A.Ein := FALSE;
   BB1_SR_K.A.B2 := FALSE;
   BB1_SR_K.A.FU := FALSE;
   BB1_SR_K.A.Req_extern_B1 := FALSE;
   BB1_SR_K.A.Req_extern_B2 := FALSE;
   BB1_SR_K.A.Dir := FALSE;
   BB1_SR_K.A.RST := FALSE;
   BB1_SR_K.A.Auf := FALSE;
   BB1_SR_K.A.Zu := FALSE;
   BB1_SR_K.A.Res9 := FALSE;
   BB1_SR_K.A.Res10 := FALSE;
   BB1_SR_K.A.Res11 := FALSE;
   BB1_SR_K.A.Res12 := FALSE;
   BB1_SR_K.A.Res13 := FALSE;
   BB1_SR_K.A.Res14 := FALSE;
   BB1_SR_K.A.Quit_extern := FALSE;
   Zulauf_AR_P1.E.Ein := FALSE;
   Zulauf_AR_P1.E.Anst := FALSE;
   Zulauf_AR_P1.E.FU := FALSE;
   Zulauf_AR_P1.E.EA := FALSE;
   Zulauf_AR_P1.E.EZ := FALSE;
   Zulauf_AR_P1.E.MS_St := FALSE;
   Zulauf_AR_P1.E.Th_St := FALSE;
   Zulauf_AR_P1.E.DMA_St := FALSE;
   Zulauf_AR_P1.E.DMZ_St := FALSE;
   Zulauf_AR_P1.E.FU_St := FALSE;
   Zulauf_AR_P1.E.TL_St := FALSE;
   Zulauf_AR_P1.E.UDr_St := FALSE;
   Zulauf_AR_P1.E.UeDr_St := FALSE;
   Zulauf_AR_P1.E.UT_St := FALSE;
   Zulauf_AR_P1.E.Le_St := FALSE;
   Zulauf_AR_P1.E.UeLM_St := FALSE;
   Zulauf_AR_P1.E.UeLE_St := FALSE;
   Zulauf_AR_P1.E.Kom_DP_St := FALSE;
   Zulauf_AR_P1.E.Kom_int_St := FALSE;
   Zulauf_AR_P1.E.int_St := FALSE;
   Zulauf_AR_P1.E.Wart_Wa := FALSE;
   Zulauf_AR_P1.E.Bed_vOrt := FALSE;
   Zulauf_AR_P1.E.Bed_Fern := TRUE;
   Zulauf_AR_P1.E.Bed_UV := FALSE;
   Zulauf_AR_P1.E.Aus := FALSE;
   Zulauf_AR_P1.E.NA := FALSE;
   Zulauf_AR_P1.E.AF_St := FALSE;
   Zulauf_AR_P1.E.Strm := FALSE;
   Zulauf_AR_P1.E.FI_St := FALSE;
   Zulauf_AR_P1.E.SA_St := FALSE;
   Zulauf_AR_P1.E.DD_St := FALSE;
   Zulauf_AR_P1.E.St := FALSE;
   Zulauf_AR_P1.A.Ein := FALSE;
   Zulauf_AR_P1.A.B2 := FALSE;
   Zulauf_AR_P1.A.FU := FALSE;
   Zulauf_AR_P1.A.Req_extern_B1 := FALSE;
   Zulauf_AR_P1.A.Req_extern_B2 := FALSE;
   Zulauf_AR_P1.A.Dir := FALSE;
   Zulauf_AR_P1.A.RST := FALSE;
   Zulauf_AR_P1.A.Auf := FALSE;
   Zulauf_AR_P1.A.Zu := FALSE;
   Zulauf_AR_P1.A.Res9 := FALSE;
   Zulauf_AR_P1.A.Res10 := FALSE;
   Zulauf_AR_P1.A.Res11 := FALSE;
   Zulauf_AR_P1.A.Res12 := FALSE;
   Zulauf_AR_P1.A.Res13 := FALSE;
   Zulauf_AR_P1.A.Res14 := FALSE;
   Zulauf_AR_P1.A.Quit_extern := FALSE;
   Zulauf_AR_P2.E.Ein := FALSE;
   Zulauf_AR_P2.E.Anst := FALSE;
   Zulauf_AR_P2.E.FU := FALSE;
   Zulauf_AR_P2.E.EA := FALSE;
   Zulauf_AR_P2.E.EZ := FALSE;
   Zulauf_AR_P2.E.MS_St := FALSE;
   Zulauf_AR_P2.E.Th_St := FALSE;
   Zulauf_AR_P2.E.DMA_St := FALSE;
   Zulauf_AR_P2.E.DMZ_St := FALSE;
   Zulauf_AR_P2.E.FU_St := FALSE;
   Zulauf_AR_P2.E.TL_St := FALSE;
   Zulauf_AR_P2.E.UDr_St := FALSE;
   Zulauf_AR_P2.E.UeDr_St := FALSE;
   Zulauf_AR_P2.E.UT_St := FALSE;
   Zulauf_AR_P2.E.Le_St := FALSE;
   Zulauf_AR_P2.E.UeLM_St := FALSE;
   Zulauf_AR_P2.E.UeLE_St := FALSE;
   Zulauf_AR_P2.E.Kom_DP_St := FALSE;
   Zulauf_AR_P2.E.Kom_int_St := FALSE;
   Zulauf_AR_P2.E.int_St := FALSE;
   Zulauf_AR_P2.E.Wart_Wa := FALSE;
   Zulauf_AR_P2.E.Bed_vOrt := FALSE;
   Zulauf_AR_P2.E.Bed_Fern := TRUE;
   Zulauf_AR_P2.E.Bed_UV := FALSE;
   Zulauf_AR_P2.E.Aus := FALSE;
   Zulauf_AR_P2.E.NA := FALSE;
   Zulauf_AR_P2.E.AF_St := FALSE;
   Zulauf_AR_P2.E.Strm := FALSE;
   Zulauf_AR_P2.E.FI_St := FALSE;
   Zulauf_AR_P2.E.SA_St := FALSE;
   Zulauf_AR_P2.E.DD_St := FALSE;
   Zulauf_AR_P2.E.St := FALSE;
   Zulauf_AR_P2.A.Ein := FALSE;
   Zulauf_AR_P2.A.B2 := FALSE;
   Zulauf_AR_P2.A.FU := FALSE;
   Zulauf_AR_P2.A.Req_extern_B1 := FALSE;
   Zulauf_AR_P2.A.Req_extern_B2 := FALSE;
   Zulauf_AR_P2.A.Dir := FALSE;
   Zulauf_AR_P2.A.RST := FALSE;
   Zulauf_AR_P2.A.Auf := FALSE;
   Zulauf_AR_P2.A.Zu := FALSE;
   Zulauf_AR_P2.A.Res9 := FALSE;
   Zulauf_AR_P2.A.Res10 := FALSE;
   Zulauf_AR_P2.A.Res11 := FALSE;
   Zulauf_AR_P2.A.Res12 := FALSE;
   Zulauf_AR_P2.A.Res13 := FALSE;
   Zulauf_AR_P2.A.Res14 := FALSE;
   Zulauf_AR_P2.A.Quit_extern := FALSE;
   Zulauf_AS.E.Ein := FALSE;
   Zulauf_AS.E.Anst := FALSE;
   Zulauf_AS.E.FU := FALSE;
   Zulauf_AS.E.EA := FALSE;
   Zulauf_AS.E.EZ := FALSE;
   Zulauf_AS.E.MS_St := FALSE;
   Zulauf_AS.E.Th_St := FALSE;
   Zulauf_AS.E.DMA_St := FALSE;
   Zulauf_AS.E.DMZ_St := FALSE;
   Zulauf_AS.E.FU_St := FALSE;
   Zulauf_AS.E.TL_St := FALSE;
   Zulauf_AS.E.UDr_St := FALSE;
   Zulauf_AS.E.UeDr_St := FALSE;
   Zulauf_AS.E.UT_St := FALSE;
   Zulauf_AS.E.Le_St := FALSE;
   Zulauf_AS.E.UeLM_St := FALSE;
   Zulauf_AS.E.UeLE_St := FALSE;
   Zulauf_AS.E.Kom_DP_St := FALSE;
   Zulauf_AS.E.Kom_int_St := FALSE;
   Zulauf_AS.E.int_St := FALSE;
   Zulauf_AS.E.Wart_Wa := FALSE;
   Zulauf_AS.E.Bed_vOrt := FALSE;
   Zulauf_AS.E.Bed_Fern := TRUE;
   Zulauf_AS.E.Bed_UV := FALSE;
   Zulauf_AS.E.Aus := FALSE;
   Zulauf_AS.E.NA := FALSE;
   Zulauf_AS.E.AF_St := TRUE;
   Zulauf_AS.E.Strm := FALSE;
   Zulauf_AS.E.FI_St := FALSE;
   Zulauf_AS.E.SA_St := FALSE;
   Zulauf_AS.E.DD_St := FALSE;
   Zulauf_AS.E.St := FALSE;
   Zulauf_AS.A.Ein := FALSE;
   Zulauf_AS.A.B2 := FALSE;
   Zulauf_AS.A.FU := FALSE;
   Zulauf_AS.A.Req_extern_B1 := FALSE;
   Zulauf_AS.A.Req_extern_B2 := FALSE;
   Zulauf_AS.A.Dir := FALSE;
   Zulauf_AS.A.RST := FALSE;
   Zulauf_AS.A.Auf := FALSE;
   Zulauf_AS.A.Zu := FALSE;
   Zulauf_AS.A.Res9 := FALSE;
   Zulauf_AS.A.Res10 := FALSE;
   Zulauf_AS.A.Res11 := FALSE;
   Zulauf_AS.A.Res12 := FALSE;
   Zulauf_AS.A.Res13 := FALSE;
   Zulauf_AS.A.Res14 := FALSE;
   Zulauf_AS.A.Quit_extern := FALSE;
   Zulauf_RA_SA.E.Ein := FALSE;
   Zulauf_RA_SA.E.Anst := FALSE;
   Zulauf_RA_SA.E.FU := FALSE;
   Zulauf_RA_SA.E.EA := FALSE;
   Zulauf_RA_SA.E.EZ := FALSE;
   Zulauf_RA_SA.E.MS_St := FALSE;
   Zulauf_RA_SA.E.Th_St := FALSE;
   Zulauf_RA_SA.E.DMA_St := FALSE;
   Zulauf_RA_SA.E.DMZ_St := FALSE;
   Zulauf_RA_SA.E.FU_St := FALSE;
   Zulauf_RA_SA.E.TL_St := FALSE;
   Zulauf_RA_SA.E.UDr_St := FALSE;
   Zulauf_RA_SA.E.UeDr_St := FALSE;
   Zulauf_RA_SA.E.UT_St := FALSE;
   Zulauf_RA_SA.E.Le_St := FALSE;
   Zulauf_RA_SA.E.UeLM_St := FALSE;
   Zulauf_RA_SA.E.UeLE_St := FALSE;
   Zulauf_RA_SA.E.Kom_DP_St := FALSE;
   Zulauf_RA_SA.E.Kom_int_St := FALSE;
   Zulauf_RA_SA.E.int_St := FALSE;
   Zulauf_RA_SA.E.Wart_Wa := FALSE;
   Zulauf_RA_SA.E.Bed_vOrt := FALSE;
   Zulauf_RA_SA.E.Bed_Fern := TRUE;
   Zulauf_RA_SA.E.Bed_UV := FALSE;
   Zulauf_RA_SA.E.Aus := FALSE;
   Zulauf_RA_SA.E.NA := FALSE;
   Zulauf_RA_SA.E.AF_St := FALSE;
   Zulauf_RA_SA.E.Strm := FALSE;
   Zulauf_RA_SA.E.FI_St := FALSE;
   Zulauf_RA_SA.E.SA_St := FALSE;
   Zulauf_RA_SA.E.DD_St := FALSE;
   Zulauf_RA_SA.E.St := FALSE;
   Zulauf_RA_SA.A.Ein := FALSE;
   Zulauf_RA_SA.A.B2 := FALSE;
   Zulauf_RA_SA.A.FU := FALSE;
   Zulauf_RA_SA.A.Req_extern_B1 := FALSE;
   Zulauf_RA_SA.A.Req_extern_B2 := FALSE;
   Zulauf_RA_SA.A.Dir := FALSE;
   Zulauf_RA_SA.A.RST := FALSE;
   Zulauf_RA_SA.A.Auf := FALSE;
   Zulauf_RA_SA.A.Zu := FALSE;
   Zulauf_RA_SA.A.Res9 := FALSE;
   Zulauf_RA_SA.A.Res10 := FALSE;
   Zulauf_RA_SA.A.Res11 := FALSE;
   Zulauf_RA_SA.A.Res12 := FALSE;
   Zulauf_RA_SA.A.Res13 := FALSE;
   Zulauf_RA_SA.A.Res14 := FALSE;
   Zulauf_RA_SA.A.Quit_extern := FALSE;
   Zulauf_RA_HZS.E.Ein := FALSE;
   Zulauf_RA_HZS.E.Anst := FALSE;
   Zulauf_RA_HZS.E.FU := FALSE;
   Zulauf_RA_HZS.E.EA := FALSE;
   Zulauf_RA_HZS.E.EZ := FALSE;
   Zulauf_RA_HZS.E.MS_St := FALSE;
   Zulauf_RA_HZS.E.Th_St := FALSE;
   Zulauf_RA_HZS.E.DMA_St := FALSE;
   Zulauf_RA_HZS.E.DMZ_St := FALSE;
   Zulauf_RA_HZS.E.FU_St := FALSE;
   Zulauf_RA_HZS.E.TL_St := FALSE;
   Zulauf_RA_HZS.E.UDr_St := FALSE;
   Zulauf_RA_HZS.E.UeDr_St := FALSE;
   Zulauf_RA_HZS.E.UT_St := FALSE;
   Zulauf_RA_HZS.E.Le_St := FALSE;
   Zulauf_RA_HZS.E.UeLM_St := FALSE;
   Zulauf_RA_HZS.E.UeLE_St := FALSE;
   Zulauf_RA_HZS.E.Kom_DP_St := FALSE;
   Zulauf_RA_HZS.E.Kom_int_St := FALSE;
   Zulauf_RA_HZS.E.int_St := FALSE;
   Zulauf_RA_HZS.E.Wart_Wa := FALSE;
   Zulauf_RA_HZS.E.Bed_vOrt := FALSE;
   Zulauf_RA_HZS.E.Bed_Fern := TRUE;
   Zulauf_RA_HZS.E.Bed_UV := FALSE;
   Zulauf_RA_HZS.E.Aus := FALSE;
   Zulauf_RA_HZS.E.NA := FALSE;
   Zulauf_RA_HZS.E.AF_St := FALSE;
   Zulauf_RA_HZS.E.Strm := FALSE;
   Zulauf_RA_HZS.E.FI_St := FALSE;
   Zulauf_RA_HZS.E.SA_St := FALSE;
   Zulauf_RA_HZS.E.DD_St := FALSE;
   Zulauf_RA_HZS.E.St := FALSE;
   Zulauf_RA_HZS.A.Ein := FALSE;
   Zulauf_RA_HZS.A.B2 := FALSE;
   Zulauf_RA_HZS.A.FU := FALSE;
   Zulauf_RA_HZS.A.Req_extern_B1 := FALSE;
   Zulauf_RA_HZS.A.Req_extern_B2 := FALSE;
   Zulauf_RA_HZS.A.Dir := FALSE;
   Zulauf_RA_HZS.A.RST := FALSE;
   Zulauf_RA_HZS.A.Auf := FALSE;
   Zulauf_RA_HZS.A.Zu := FALSE;
   Zulauf_RA_HZS.A.Res9 := FALSE;
   Zulauf_RA_HZS.A.Res10 := FALSE;
   Zulauf_RA_HZS.A.Res11 := FALSE;
   Zulauf_RA_HZS.A.Res12 := FALSE;
   Zulauf_RA_HZS.A.Res13 := FALSE;
   Zulauf_RA_HZS.A.Res14 := FALSE;
   Zulauf_RA_HZS.A.Quit_extern := FALSE;
   Zulauf_RA_VKS.E.Ein := FALSE;
   Zulauf_RA_VKS.E.Anst := FALSE;
   Zulauf_RA_VKS.E.FU := FALSE;
   Zulauf_RA_VKS.E.EA := FALSE;
   Zulauf_RA_VKS.E.EZ := FALSE;
   Zulauf_RA_VKS.E.MS_St := FALSE;
   Zulauf_RA_VKS.E.Th_St := FALSE;
   Zulauf_RA_VKS.E.DMA_St := FALSE;
   Zulauf_RA_VKS.E.DMZ_St := FALSE;
   Zulauf_RA_VKS.E.FU_St := FALSE;
   Zulauf_RA_VKS.E.TL_St := FALSE;
   Zulauf_RA_VKS.E.UDr_St := FALSE;
   Zulauf_RA_VKS.E.UeDr_St := FALSE;
   Zulauf_RA_VKS.E.UT_St := FALSE;
   Zulauf_RA_VKS.E.Le_St := FALSE;
   Zulauf_RA_VKS.E.UeLM_St := FALSE;
   Zulauf_RA_VKS.E.UeLE_St := FALSE;
   Zulauf_RA_VKS.E.Kom_DP_St := FALSE;
   Zulauf_RA_VKS.E.Kom_int_St := FALSE;
   Zulauf_RA_VKS.E.int_St := FALSE;
   Zulauf_RA_VKS.E.Wart_Wa := FALSE;
   Zulauf_RA_VKS.E.Bed_vOrt := FALSE;
   Zulauf_RA_VKS.E.Bed_Fern := TRUE;
   Zulauf_RA_VKS.E.Bed_UV := FALSE;
   Zulauf_RA_VKS.E.Aus := FALSE;
   Zulauf_RA_VKS.E.NA := FALSE;
   Zulauf_RA_VKS.E.AF_St := FALSE;
   Zulauf_RA_VKS.E.Strm := FALSE;
   Zulauf_RA_VKS.E.FI_St := FALSE;
   Zulauf_RA_VKS.E.SA_St := FALSE;
   Zulauf_RA_VKS.E.DD_St := FALSE;
   Zulauf_RA_VKS.E.St := FALSE;
   Zulauf_RA_VKS.A.Ein := FALSE;
   Zulauf_RA_VKS.A.B2 := FALSE;
   Zulauf_RA_VKS.A.FU := FALSE;
   Zulauf_RA_VKS.A.Req_extern_B1 := FALSE;
   Zulauf_RA_VKS.A.Req_extern_B2 := FALSE;
   Zulauf_RA_VKS.A.Dir := FALSE;
   Zulauf_RA_VKS.A.RST := FALSE;
   Zulauf_RA_VKS.A.Auf := FALSE;
   Zulauf_RA_VKS.A.Zu := FALSE;
   Zulauf_RA_VKS.A.Res9 := FALSE;
   Zulauf_RA_VKS.A.Res10 := FALSE;
   Zulauf_RA_VKS.A.Res11 := FALSE;
   Zulauf_RA_VKS.A.Res12 := FALSE;
   Zulauf_RA_VKS.A.Res13 := FALSE;
   Zulauf_RA_VKS.A.Res14 := FALSE;
   Zulauf_RA_VKS.A.Quit_extern := FALSE;
   Zulauf_RA_V.E.Ein := TRUE;
   Zulauf_RA_V.E.Anst := FALSE;
   Zulauf_RA_V.E.FU := FALSE;
   Zulauf_RA_V.E.EA := FALSE;
   Zulauf_RA_V.E.EZ := FALSE;
   Zulauf_RA_V.E.MS_St := FALSE;
   Zulauf_RA_V.E.Th_St := FALSE;
   Zulauf_RA_V.E.DMA_St := FALSE;
   Zulauf_RA_V.E.DMZ_St := FALSE;
   Zulauf_RA_V.E.FU_St := FALSE;
   Zulauf_RA_V.E.TL_St := FALSE;
   Zulauf_RA_V.E.UDr_St := FALSE;
   Zulauf_RA_V.E.UeDr_St := FALSE;
   Zulauf_RA_V.E.UT_St := FALSE;
   Zulauf_RA_V.E.Le_St := FALSE;
   Zulauf_RA_V.E.UeLM_St := FALSE;
   Zulauf_RA_V.E.UeLE_St := FALSE;
   Zulauf_RA_V.E.Kom_DP_St := FALSE;
   Zulauf_RA_V.E.Kom_int_St := FALSE;
   Zulauf_RA_V.E.int_St := FALSE;
   Zulauf_RA_V.E.Wart_Wa := FALSE;
   Zulauf_RA_V.E.Bed_vOrt := FALSE;
   Zulauf_RA_V.E.Bed_Fern := TRUE;
   Zulauf_RA_V.E.Bed_UV := FALSE;
   Zulauf_RA_V.E.Aus := FALSE;
   Zulauf_RA_V.E.NA := FALSE;
   Zulauf_RA_V.E.AF_St := FALSE;
   Zulauf_RA_V.E.Strm := FALSE;
   Zulauf_RA_V.E.FI_St := FALSE;
   Zulauf_RA_V.E.SA_St := FALSE;
   Zulauf_RA_V.E.DD_St := FALSE;
   Zulauf_RA_V.E.St := FALSE;
   Zulauf_RA_V.A.Ein := FALSE;
   Zulauf_RA_V.A.B2 := FALSE;
   Zulauf_RA_V.A.FU := FALSE;
   Zulauf_RA_V.A.Req_extern_B1 := FALSE;
   Zulauf_RA_V.A.Req_extern_B2 := FALSE;
   Zulauf_RA_V.A.Dir := FALSE;
   Zulauf_RA_V.A.RST := FALSE;
   Zulauf_RA_V.A.Auf := FALSE;
   Zulauf_RA_V.A.Zu := FALSE;
   Zulauf_RA_V.A.Res9 := FALSE;
   Zulauf_RA_V.A.Res10 := FALSE;
   Zulauf_RA_V.A.Res11 := FALSE;
   Zulauf_RA_V.A.Res12 := FALSE;
   Zulauf_RA_V.A.Res13 := FALSE;
   Zulauf_RA_V.A.Res14 := FALSE;
   Zulauf_RA_V.A.Quit_extern := FALSE;
   Zulauf_RA_RP.E.Ein := FALSE;
   Zulauf_RA_RP.E.Anst := FALSE;
   Zulauf_RA_RP.E.FU := FALSE;
   Zulauf_RA_RP.E.EA := FALSE;
   Zulauf_RA_RP.E.EZ := FALSE;
   Zulauf_RA_RP.E.MS_St := FALSE;
   Zulauf_RA_RP.E.Th_St := FALSE;
   Zulauf_RA_RP.E.DMA_St := FALSE;
   Zulauf_RA_RP.E.DMZ_St := FALSE;
   Zulauf_RA_RP.E.FU_St := FALSE;
   Zulauf_RA_RP.E.TL_St := FALSE;
   Zulauf_RA_RP.E.UDr_St := FALSE;
   Zulauf_RA_RP.E.UeDr_St := FALSE;
   Zulauf_RA_RP.E.UT_St := FALSE;
   Zulauf_RA_RP.E.Le_St := FALSE;
   Zulauf_RA_RP.E.UeLM_St := FALSE;
   Zulauf_RA_RP.E.UeLE_St := FALSE;
   Zulauf_RA_RP.E.Kom_DP_St := FALSE;
   Zulauf_RA_RP.E.Kom_int_St := FALSE;
   Zulauf_RA_RP.E.int_St := FALSE;
   Zulauf_RA_RP.E.Wart_Wa := FALSE;
   Zulauf_RA_RP.E.Bed_vOrt := FALSE;
   Zulauf_RA_RP.E.Bed_Fern := TRUE;
   Zulauf_RA_RP.E.Bed_UV := FALSE;
   Zulauf_RA_RP.E.Aus := FALSE;
   Zulauf_RA_RP.E.NA := FALSE;
   Zulauf_RA_RP.E.AF_St := FALSE;
   Zulauf_RA_RP.E.Strm := FALSE;
   Zulauf_RA_RP.E.FI_St := FALSE;
   Zulauf_RA_RP.E.SA_St := FALSE;
   Zulauf_RA_RP.E.DD_St := FALSE;
   Zulauf_RA_RP.E.St := FALSE;
   Zulauf_RA_RP.A.Ein := FALSE;
   Zulauf_RA_RP.A.B2 := FALSE;
   Zulauf_RA_RP.A.FU := FALSE;
   Zulauf_RA_RP.A.Req_extern_B1 := FALSE;
   Zulauf_RA_RP.A.Req_extern_B2 := FALSE;
   Zulauf_RA_RP.A.Dir := FALSE;
   Zulauf_RA_RP.A.RST := FALSE;
   Zulauf_RA_RP.A.Auf := FALSE;
   Zulauf_RA_RP.A.Zu := FALSE;
   Zulauf_RA_RP.A.Res9 := FALSE;
   Zulauf_RA_RP.A.Res10 := FALSE;
   Zulauf_RA_RP.A.Res11 := FALSE;
   Zulauf_RA_RP.A.Res12 := FALSE;
   Zulauf_RA_RP.A.Res13 := FALSE;
   Zulauf_RA_RP.A.Res14 := FALSE;
   Zulauf_RA_RP.A.Quit_extern := FALSE;
   Zulauf_RA_FP.E.Ein := FALSE;
   Zulauf_RA_FP.E.Anst := FALSE;
   Zulauf_RA_FP.E.FU := FALSE;
   Zulauf_RA_FP.E.EA := FALSE;
   Zulauf_RA_FP.E.EZ := FALSE;
   Zulauf_RA_FP.E.MS_St := FALSE;
   Zulauf_RA_FP.E.Th_St := FALSE;
   Zulauf_RA_FP.E.DMA_St := FALSE;
   Zulauf_RA_FP.E.DMZ_St := FALSE;
   Zulauf_RA_FP.E.FU_St := FALSE;
   Zulauf_RA_FP.E.TL_St := FALSE;
   Zulauf_RA_FP.E.UDr_St := FALSE;
   Zulauf_RA_FP.E.UeDr_St := FALSE;
   Zulauf_RA_FP.E.UT_St := FALSE;
   Zulauf_RA_FP.E.Le_St := FALSE;
   Zulauf_RA_FP.E.UeLM_St := FALSE;
   Zulauf_RA_FP.E.UeLE_St := FALSE;
   Zulauf_RA_FP.E.Kom_DP_St := FALSE;
   Zulauf_RA_FP.E.Kom_int_St := FALSE;
   Zulauf_RA_FP.E.int_St := FALSE;
   Zulauf_RA_FP.E.Wart_Wa := FALSE;
   Zulauf_RA_FP.E.Bed_vOrt := FALSE;
   Zulauf_RA_FP.E.Bed_Fern := TRUE;
   Zulauf_RA_FP.E.Bed_UV := FALSE;
   Zulauf_RA_FP.E.Aus := FALSE;
   Zulauf_RA_FP.E.NA := FALSE;
   Zulauf_RA_FP.E.AF_St := FALSE;
   Zulauf_RA_FP.E.Strm := FALSE;
   Zulauf_RA_FP.E.FI_St := FALSE;
   Zulauf_RA_FP.E.SA_St := FALSE;
   Zulauf_RA_FP.E.DD_St := FALSE;
   Zulauf_RA_FP.E.St := FALSE;
   Zulauf_RA_FP.A.Ein := FALSE;
   Zulauf_RA_FP.A.B2 := FALSE;
   Zulauf_RA_FP.A.FU := FALSE;
   Zulauf_RA_FP.A.Req_extern_B1 := FALSE;
   Zulauf_RA_FP.A.Req_extern_B2 := FALSE;
   Zulauf_RA_FP.A.Dir := FALSE;
   Zulauf_RA_FP.A.RST := FALSE;
   Zulauf_RA_FP.A.Auf := FALSE;
   Zulauf_RA_FP.A.Zu := FALSE;
   Zulauf_RA_FP.A.Res9 := FALSE;
   Zulauf_RA_FP.A.Res10 := FALSE;
   Zulauf_RA_FP.A.Res11 := FALSE;
   Zulauf_RA_FP.A.Res12 := FALSE;
   Zulauf_RA_FP.A.Res13 := FALSE;
   Zulauf_RA_FP.A.Res14 := FALSE;
   Zulauf_RA_FP.A.Quit_extern := FALSE;
   Schlamm_BP.E.Ein := FALSE;
   Schlamm_BP.E.Anst := FALSE;
   Schlamm_BP.E.FU := FALSE;
   Schlamm_BP.E.EA := FALSE;
   Schlamm_BP.E.EZ := FALSE;
   Schlamm_BP.E.MS_St := FALSE;
   Schlamm_BP.E.Th_St := FALSE;
   Schlamm_BP.E.DMA_St := FALSE;
   Schlamm_BP.E.DMZ_St := FALSE;
   Schlamm_BP.E.FU_St := FALSE;
   Schlamm_BP.E.TL_St := FALSE;
   Schlamm_BP.E.UDr_St := FALSE;
   Schlamm_BP.E.UeDr_St := FALSE;
   Schlamm_BP.E.UT_St := FALSE;
   Schlamm_BP.E.Le_St := FALSE;
   Schlamm_BP.E.UeLM_St := FALSE;
   Schlamm_BP.E.UeLE_St := FALSE;
   Schlamm_BP.E.Kom_DP_St := FALSE;
   Schlamm_BP.E.Kom_int_St := FALSE;
   Schlamm_BP.E.int_St := FALSE;
   Schlamm_BP.E.Wart_Wa := FALSE;
   Schlamm_BP.E.Bed_vOrt := FALSE;
   Schlamm_BP.E.Bed_Fern := TRUE;
   Schlamm_BP.E.Bed_UV := FALSE;
   Schlamm_BP.E.Aus := FALSE;
   Schlamm_BP.E.NA := FALSE;
   Schlamm_BP.E.AF_St := FALSE;
   Schlamm_BP.E.Strm := FALSE;
   Schlamm_BP.E.FI_St := FALSE;
   Schlamm_BP.E.SA_St := FALSE;
   Schlamm_BP.E.DD_St := FALSE;
   Schlamm_BP.E.St := FALSE;
   Schlamm_BP.A.Ein := FALSE;
   Schlamm_BP.A.B2 := FALSE;
   Schlamm_BP.A.FU := FALSE;
   Schlamm_BP.A.Req_extern_B1 := FALSE;
   Schlamm_BP.A.Req_extern_B2 := FALSE;
   Schlamm_BP.A.Dir := FALSE;
   Schlamm_BP.A.RST := FALSE;
   Schlamm_BP.A.Auf := FALSE;
   Schlamm_BP.A.Zu := FALSE;
   Schlamm_BP.A.Res9 := FALSE;
   Schlamm_BP.A.Res10 := FALSE;
   Schlamm_BP.A.Res11 := FALSE;
   Schlamm_BP.A.Res12 := FALSE;
   Schlamm_BP.A.Res13 := FALSE;
   Schlamm_BP.A.Res14 := FALSE;
   Schlamm_BP.A.Quit_extern := FALSE;
   Truebwasser_P1.E.Ein := FALSE;
   Truebwasser_P1.E.Anst := FALSE;
   Truebwasser_P1.E.FU := FALSE;
   Truebwasser_P1.E.EA := FALSE;
   Truebwasser_P1.E.EZ := FALSE;
   Truebwasser_P1.E.MS_St := FALSE;
   Truebwasser_P1.E.Th_St := FALSE;
   Truebwasser_P1.E.DMA_St := FALSE;
   Truebwasser_P1.E.DMZ_St := FALSE;
   Truebwasser_P1.E.FU_St := FALSE;
   Truebwasser_P1.E.TL_St := FALSE;
   Truebwasser_P1.E.UDr_St := FALSE;
   Truebwasser_P1.E.UeDr_St := FALSE;
   Truebwasser_P1.E.UT_St := FALSE;
   Truebwasser_P1.E.Le_St := FALSE;
   Truebwasser_P1.E.UeLM_St := FALSE;
   Truebwasser_P1.E.UeLE_St := FALSE;
   Truebwasser_P1.E.Kom_DP_St := FALSE;
   Truebwasser_P1.E.Kom_int_St := FALSE;
   Truebwasser_P1.E.int_St := FALSE;
   Truebwasser_P1.E.Wart_Wa := FALSE;
   Truebwasser_P1.E.Bed_vOrt := FALSE;
   Truebwasser_P1.E.Bed_Fern := FALSE;
   Truebwasser_P1.E.Bed_UV := FALSE;
   Truebwasser_P1.E.Aus := FALSE;
   Truebwasser_P1.E.NA := FALSE;
   Truebwasser_P1.E.AF_St := FALSE;
   Truebwasser_P1.E.Strm := FALSE;
   Truebwasser_P1.E.FI_St := FALSE;
   Truebwasser_P1.E.SA_St := FALSE;
   Truebwasser_P1.E.DD_St := FALSE;
   Truebwasser_P1.E.St := FALSE;
   Truebwasser_P1.A.Ein := FALSE;
   Truebwasser_P1.A.B2 := FALSE;
   Truebwasser_P1.A.FU := FALSE;
   Truebwasser_P1.A.Req_extern_B1 := FALSE;
   Truebwasser_P1.A.Req_extern_B2 := FALSE;
   Truebwasser_P1.A.Dir := FALSE;
   Truebwasser_P1.A.RST := FALSE;
   Truebwasser_P1.A.Auf := FALSE;
   Truebwasser_P1.A.Zu := FALSE;
   Truebwasser_P1.A.Res9 := FALSE;
   Truebwasser_P1.A.Res10 := FALSE;
   Truebwasser_P1.A.Res11 := FALSE;
   Truebwasser_P1.A.Res12 := FALSE;
   Truebwasser_P1.A.Res13 := FALSE;
   Truebwasser_P1.A.Res14 := FALSE;
   Truebwasser_P1.A.Quit_extern := FALSE;
   Truebwasser_P2.E.Ein := TRUE;
   Truebwasser_P2.E.Anst := FALSE;
   Truebwasser_P2.E.FU := FALSE;
   Truebwasser_P2.E.EA := FALSE;
   Truebwasser_P2.E.EZ := FALSE;
   Truebwasser_P2.E.MS_St := FALSE;
   Truebwasser_P2.E.Th_St := FALSE;
   Truebwasser_P2.E.DMA_St := FALSE;
   Truebwasser_P2.E.DMZ_St := FALSE;
   Truebwasser_P2.E.FU_St := FALSE;
   Truebwasser_P2.E.TL_St := FALSE;
   Truebwasser_P2.E.UDr_St := FALSE;
   Truebwasser_P2.E.UeDr_St := FALSE;
   Truebwasser_P2.E.UT_St := FALSE;
   Truebwasser_P2.E.Le_St := FALSE;
   Truebwasser_P2.E.UeLM_St := FALSE;
   Truebwasser_P2.E.UeLE_St := FALSE;
   Truebwasser_P2.E.Kom_DP_St := FALSE;
   Truebwasser_P2.E.Kom_int_St := FALSE;
   Truebwasser_P2.E.int_St := FALSE;
   Truebwasser_P2.E.Wart_Wa := FALSE;
   Truebwasser_P2.E.Bed_vOrt := FALSE;
   Truebwasser_P2.E.Bed_Fern := TRUE;
   Truebwasser_P2.E.Bed_UV := FALSE;
   Truebwasser_P2.E.Aus := FALSE;
   Truebwasser_P2.E.NA := FALSE;
   Truebwasser_P2.E.AF_St := FALSE;
   Truebwasser_P2.E.Strm := FALSE;
   Truebwasser_P2.E.FI_St := FALSE;
   Truebwasser_P2.E.SA_St := FALSE;
   Truebwasser_P2.E.DD_St := FALSE;
   Truebwasser_P2.E.St := FALSE;
   Truebwasser_P2.A.Ein := TRUE;
   Truebwasser_P2.A.B2 := FALSE;
   Truebwasser_P2.A.FU := FALSE;
   Truebwasser_P2.A.Req_extern_B1 := TRUE;
   Truebwasser_P2.A.Req_extern_B2 := FALSE;
   Truebwasser_P2.A.Dir := FALSE;
   Truebwasser_P2.A.RST := FALSE;
   Truebwasser_P2.A.Auf := FALSE;
   Truebwasser_P2.A.Zu := FALSE;
   Truebwasser_P2.A.Res9 := FALSE;
   Truebwasser_P2.A.Res10 := FALSE;
   Truebwasser_P2.A.Res11 := FALSE;
   Truebwasser_P2.A.Res12 := FALSE;
   Truebwasser_P2.A.Res13 := FALSE;
   Truebwasser_P2.A.Res14 := FALSE;
   Truebwasser_P2.A.Quit_extern := FALSE;
   Schlamm_AS.E.Ein := FALSE;
   Schlamm_AS.E.Anst := FALSE;
   Schlamm_AS.E.FU := FALSE;
   Schlamm_AS.E.EA := FALSE;
   Schlamm_AS.E.EZ := TRUE;
   Schlamm_AS.E.MS_St := FALSE;
   Schlamm_AS.E.Th_St := FALSE;
   Schlamm_AS.E.DMA_St := FALSE;
   Schlamm_AS.E.DMZ_St := FALSE;
   Schlamm_AS.E.FU_St := FALSE;
   Schlamm_AS.E.TL_St := FALSE;
   Schlamm_AS.E.UDr_St := FALSE;
   Schlamm_AS.E.UeDr_St := FALSE;
   Schlamm_AS.E.UT_St := FALSE;
   Schlamm_AS.E.Le_St := FALSE;
   Schlamm_AS.E.UeLM_St := FALSE;
   Schlamm_AS.E.UeLE_St := FALSE;
   Schlamm_AS.E.Kom_DP_St := FALSE;
   Schlamm_AS.E.Kom_int_St := FALSE;
   Schlamm_AS.E.int_St := FALSE;
   Schlamm_AS.E.Wart_Wa := FALSE;
   Schlamm_AS.E.Bed_vOrt := FALSE;
   Schlamm_AS.E.Bed_Fern := TRUE;
   Schlamm_AS.E.Bed_UV := FALSE;
   Schlamm_AS.E.Aus := FALSE;
   Schlamm_AS.E.NA := FALSE;
   Schlamm_AS.E.AF_St := FALSE;
   Schlamm_AS.E.Strm := FALSE;
   Schlamm_AS.E.FI_St := FALSE;
   Schlamm_AS.E.SA_St := FALSE;
   Schlamm_AS.E.DD_St := FALSE;
   Schlamm_AS.E.St := FALSE;
   Schlamm_AS.A.Ein := FALSE;
   Schlamm_AS.A.B2 := FALSE;
   Schlamm_AS.A.FU := FALSE;
   Schlamm_AS.A.Req_extern_B1 := FALSE;
   Schlamm_AS.A.Req_extern_B2 := FALSE;
   Schlamm_AS.A.Dir := FALSE;
   Schlamm_AS.A.RST := FALSE;
   Schlamm_AS.A.Auf := FALSE;
   Schlamm_AS.A.Zu := FALSE;
   Schlamm_AS.A.Res9 := FALSE;
   Schlamm_AS.A.Res10 := FALSE;
   Schlamm_AS.A.Res11 := FALSE;
   Schlamm_AS.A.Res12 := FALSE;
   Schlamm_AS.A.Res13 := FALSE;
   Schlamm_AS.A.Res14 := FALSE;
   Schlamm_AS.A.Quit_extern := FALSE;
   BB2_SR_K.E.Ein := FALSE;
   BB2_SR_K.E.Anst := FALSE;
   BB2_SR_K.E.FU := FALSE;
   BB2_SR_K.E.EA := FALSE;
   BB2_SR_K.E.EZ := FALSE;
   BB2_SR_K.E.MS_St := FALSE;
   BB2_SR_K.E.Th_St := FALSE;
   BB2_SR_K.E.DMA_St := FALSE;
   BB2_SR_K.E.DMZ_St := FALSE;
   BB2_SR_K.E.FU_St := FALSE;
   BB2_SR_K.E.TL_St := FALSE;
   BB2_SR_K.E.UDr_St := FALSE;
   BB2_SR_K.E.UeDr_St := FALSE;
   BB2_SR_K.E.UT_St := FALSE;
   BB2_SR_K.E.Le_St := FALSE;
   BB2_SR_K.E.UeLM_St := FALSE;
   BB2_SR_K.E.UeLE_St := FALSE;
   BB2_SR_K.E.Kom_DP_St := FALSE;
   BB2_SR_K.E.Kom_int_St := FALSE;
   BB2_SR_K.E.int_St := FALSE;
   BB2_SR_K.E.Wart_Wa := FALSE;
   BB2_SR_K.E.Bed_vOrt := FALSE;
   BB2_SR_K.E.Bed_Fern := TRUE;
   BB2_SR_K.E.Bed_UV := FALSE;
   BB2_SR_K.E.Aus := FALSE;
   BB2_SR_K.E.NA := FALSE;
   BB2_SR_K.E.AF_St := FALSE;
   BB2_SR_K.E.Strm := FALSE;
   BB2_SR_K.E.FI_St := FALSE;
   BB2_SR_K.E.SA_St := FALSE;
   BB2_SR_K.E.DD_St := FALSE;
   BB2_SR_K.E.St := FALSE;
   BB2_SR_K.A.Ein := FALSE;
   BB2_SR_K.A.B2 := FALSE;
   BB2_SR_K.A.FU := FALSE;
   BB2_SR_K.A.Req_extern_B1 := FALSE;
   BB2_SR_K.A.Req_extern_B2 := FALSE;
   BB2_SR_K.A.Dir := FALSE;
   BB2_SR_K.A.RST := FALSE;
   BB2_SR_K.A.Auf := FALSE;
   BB2_SR_K.A.Zu := FALSE;
   BB2_SR_K.A.Res9 := FALSE;
   BB2_SR_K.A.Res10 := FALSE;
   BB2_SR_K.A.Res11 := FALSE;
   BB2_SR_K.A.Res12 := FALSE;
   BB2_SR_K.A.Res13 := FALSE;
   BB2_SR_K.A.Res14 := FALSE;
   BB2_SR_K.A.Quit_extern := FALSE;

END_DATA_BLOCK

DATA_BLOCK "DB114_MW_Meld"
{ S7_Optimized_Access := 'FALSE' }
VERSION : 0.1
NON_RETAIN
   STRUCT
      Zulauf_AR_Niv : "T_MW_MELD";   // Zulauf - Pumpwerk "Alter Rechen" - Niveau
      Zulauf_AR_Temp : "T_MW_MELD";   // Zulauf - Pumpwerk "Alter Rechen" - Temperatur
      Zulauf_AR_DF : "T_MW_MELD";   // Zulauf - Pumpwerk "Alter Rechen" - Durchfluss
      BB1_AS1_SS : "T_MW_MELD";   // Becken 1 - Ablaufschieber 1 - Schieberstellung
      BB1_AS2_SS : "T_MW_MELD";   // Becken 1 - Ablaufschieber 2 - Schieberstellung
      BB2_AS1_SS : "T_MW_MELD";   // Becken 2 - Ablaufschieber 1 - Schieberstellung
      BB2_AS2_SS : "T_MW_MELD";   // Becken 2 - Ablaufschieber 2 - Schieberstellung
      BB1_O2 : "T_MW_MELD";   // Becken 1 - O2-Gehalt
      BB1_Temp : "T_MW_MELD";   // Becken 1 - Temperatur
      BB2_O2 : "T_MW_MELD";   // Becken 2 - O2-Gehalt
      BB2_Temp : "T_MW_MELD";   // Becken 2 - Temperatur
      BB1_DF : "T_MW_MELD";   // Becken 1 - Ablauf - Durchfluss
      BB2_DF : "T_MW_MELD";   // Becken 2 - Ablauf - Durchfluss
      Zulauf_Niv : "T_MW_MELD";   // Zulauf - Vorlagebehälter - Niveau
      Zulauf_DF : "T_MW_MELD";   // Zulauf - Rechen - Durchfluss
      Verteiler_pH : "T_MW_MELD";   // Zulauf - Verteiler - pH-Wert
      Verteiler_O2 : "T_MW_MELD";   // Zulauf - Verteiler  - O2-Gehalt
      Verteiler_Temp : "T_MW_MELD";   // Zulauf - Verteiler - Temperatur
      BB_UeSS_DF : "T_MW_MELD";   // Becken 1+2 - Ablauf ÜSS - Durchfluss
      Ablauf_DF : "T_MW_MELD";   // Ablauf - Durchfluss
      Ablauf_pH : "T_MW_MELD";   // Ablauf - pH-Wert
      Ablauf_O2 : "T_MW_MELD";   // Ablauf - O2-Gehalt
      Ablauf_Temp : "T_MW_MELD";   // Ablauf - Temperatur
      Schlamm_ED_Niv : "T_MW_MELD";   // Schlamm - Eindicker - Niveau
      Schlamm_Besch_Niv : "T_MW_MELD";   // Schlamm - Beschickung - Niveau
      Schlamm_Besch_DF : "T_MW_MELD";   // Schlamm - Beschickung - Durchfluss
      Truebwasser_Niv : "T_MW_MELD";   // Trübwasserpumpwerk - Niveau
      Truebwasser_DF : "T_MW_MELD";   // Trübwasserpumpwerk - Durchfluss
      Zulauf_SF_Niv : "T_MW_MELD";   // Zulauf - Sandfang - Niveau
      Ablauf_NOx : "T_MW_MELD";   // Ablauf - Dortmundbrunnen - Nitratmessung
      Ablauf_PO4 : "T_MW_MELD";   // Ablauf - Dortmundbrunnen - Phosphatmessung
      Umwelt_WG : "T_MW_MELD";   // Wetterstation - Windgeschwindigkeit
      Umwelt_WR : "T_MW_MELD";   // Wetterstation - Windrichtung
      Umwelt_LDr : "T_MW_MELD";   // Wetterstation - Luftdruck
      Umwelt_LF : "T_MW_MELD";   // Wetterstation - Luftfeuchtigkeit
      Umwelt_T : "T_MW_MELD";   // Wetterstation - Temperatur
      Ablauf_LF : "T_MW_MELD";   // Ablauf - Leitfähigkeit
   END_STRUCT;


